// Writing clear text for field description
IF (nMemoryBank = 0) THEN
	aMemoryBank[0].sName := ' Address of last accessible memory location (read only)';
	aMemoryBank[1].sName := ' Reserved-not implemented ';
	aMemoryBank[2].sName := ' Number of last accessible memory bank (read only)';
	aMemoryBank[3].sName := ' GTIN byte 0 (MSB) (read only)';
	aMemoryBank[4].sName := ' GTIN byte 1 (read only)';
	aMemoryBank[5].sName := ' GTIN byte 2 (read only)';
	aMemoryBank[6].sName := ' GTIN byte 3 (read only)';
	aMemoryBank[7].sName := ' GTIN byte 4 (read only)';
	aMemoryBank[8].sName := ' GTIN byte 5 (LSB) (read only)';
	aMemoryBank[9].sName := ' Firmware Version (major) (read only)';
	aMemoryBank[10].sName := ' Firmware Version (m)(read only)';
	aMemoryBank[11].sName := ' Identification number byte 0 (MSB) (read only)';
	aMemoryBank[12].sName := ' Identification number byte 1 (read only)';
	aMemoryBank[13].sName := ' Identification number byte 2 (read only)';
	aMemoryBank[14].sName := ' Identification number byte 3 (read only)';
	aMemoryBank[15].sName := ' Identification number byte 4 (read only)';
	aMemoryBank[16].sName := ' Identification number byte 5 (read only)';
	aMemoryBank[17].sName := ' Identification number byte 6 (read only)';
	aMemoryBank[18].sName := ' Identification number byte 7 (LSB) (read only)';
	aMemoryBank[19].sName := ' Hardware version (major)(read only)'; 
	aMemoryBank[20].sName := ' Hardware version (minor)(read only)'; 
	aMemoryBank[21].sName := ' 101 version number (read only)';
	aMemoryBank[22].sName := ' 102 version number of all integrated control gear (read only)';
	aMemoryBank[23].sName := ' 103 version number of all integrates control devices (read only)';
	aMemoryBank[24].sName := ' Number of logical control device units in the bus unit (read only)';
	aMemoryBank[25].sName := ' Number of logical control gear units in the bus unit(read only)';
	aMemoryBank[26].sName := ' Index number of this logical control gear unit (read only)';
END_IF
IF (nMemoryBank = 1) THEN
	aMemoryBank[0].sName := ' Address of last accessible memory location (read only)';
	aMemoryBank[1].sName := ' Indicator byte (manufacturer defined) ';
	aMemoryBank[2].sName := ' Memory bank 1 lock byte';
	aMemoryBank[3].sName := ' OEM GTIN byte 0 (MSB) (read only)';
	aMemoryBank[4].sName := ' OEM GTIN byte 1 (read only)';
	aMemoryBank[5].sName := ' OEM GTIN byte 2 (read only)';
	aMemoryBank[6].sName := ' OEM GTIN byte 3 (read only)';
	aMemoryBank[7].sName := ' OEM GTIN byte 4 (read only)';
	aMemoryBank[8].sName := ' OEM GTIN byte 5 (LSB) (read only)';
	aMemoryBank[9].sName := ' OEM identification number byte 0 (MSB)';
	aMemoryBank[10].sName := ' OEM identification number byte 1';
	aMemoryBank[11].sName := ' OEM identification number byte 2';
	aMemoryBank[12].sName := ' OEM identification number byte 3';
	aMemoryBank[13].sName := ' OEM identification number byte 4';
	aMemoryBank[14].sName := ' OEM identification number byte 5';
	aMemoryBank[15].sName := ' OEM identification number byte 6';
	aMemoryBank[16].sName := ' OEM identification number byte 7 (LSB)';
END_IF
IF (nMemoryBank >= 1) THEN
	aMemoryBank[17].sName := ' Additional control gear information (lockable)';
	aMemoryBank[18].sName := ' Additional control gear information (lockable)';
	aMemoryBank[19].sName := ' Additional control gear information (lockable)';
	aMemoryBank[20].sName := ' Additional control gear information (lockable)';
	aMemoryBank[21].sName := ' Additional control gear information (lockable)';
	aMemoryBank[22].sName := ' Additional control gear information (lockable)';
	aMemoryBank[23].sName := ' Additional control gear information (lockable)';
	aMemoryBank[24].sName := ' Additional control gear information (lockable)';
	aMemoryBank[25].sName := ' Additional control gear information (lockable)';
	aMemoryBank[26].sName := ' Additional control gear information (lockable)';
	aMemoryBank[27].sName := ' Additional control gear information (lockable)';
	aMemoryBank[28].sName := ' Additional control gear information (lockable)';
	aMemoryBank[29].sName := ' Additional control gear information (lockable)';
	aMemoryBank[30].sName := ' Additional control gear information (lockable)';
	aMemoryBank[31].sName := ' Additional control gear information (lockable)';
	aMemoryBank[32].sName := ' Additional control gear information (lockable)';
	aMemoryBank[33].sName := ' Additional control gear information (lockable)';
	aMemoryBank[34].sName := ' Additional control gear information (lockable)';
	aMemoryBank[35].sName := ' Additional control gear information (lockable)';
	aMemoryBank[36].sName := ' Additional control gear information (lockable)';
	aMemoryBank[37].sName := ' Additional control gear information (lockable)';
	aMemoryBank[38].sName := ' Additional control gear information (lockable)';
	aMemoryBank[39].sName := ' Additional control gear information (lockable)';
	aMemoryBank[40].sName := ' Additional control gear information (lockable)';
	aMemoryBank[41].sName := ' Additional control gear information (lockable)';
	aMemoryBank[42].sName := ' Additional control gear information (lockable)';
	aMemoryBank[42].sName := ' Additional control gear information (lockable)';
	aMemoryBank[44].sName := ' Additional control gear information (lockable)';
	aMemoryBank[45].sName := ' Additional control gear information (lockable)';
	aMemoryBank[46].sName := ' Additional control gear information (lockable)';
	aMemoryBank[47].sName := ' Additional control gear information (lockable)';
	aMemoryBank[48].sName := ' Additional control gear information (lockable)';
	aMemoryBank[49].sName := ' Additional control gear information (lockable)';
	aMemoryBank[50].sName := ' Additional control gear information (lockable)';
	aMemoryBank[51].sName := ' Additional control gear information (lockable)';
	aMemoryBank[52].sName := ' Additional control gear information (lockable)';
	aMemoryBank[53].sName := ' Additional control gear information (lockable)';
	aMemoryBank[54].sName := ' Additional control gear information (lockable)';
	aMemoryBank[55].sName := ' Additional control gear information (lockable)';
	aMemoryBank[56].sName := ' Additional control gear information (lockable)';
	aMemoryBank[57].sName := ' Additional control gear information (lockable)';
	aMemoryBank[58].sName := ' Additional control gear information (lockable)';
	aMemoryBank[59].sName := ' Additional control gear information (lockable)';
	aMemoryBank[60].sName := ' Additional control gear information (lockable)';
	aMemoryBank[61].sName := ' Additional control gear information (lockable)';
	aMemoryBank[62].sName := ' Additional control gear information (lockable)';
	aMemoryBank[63].sName := ' Additional control gear information (lockable)';
	aMemoryBank[64].sName := ' Additional control gear information (lockable)';
	aMemoryBank[65].sName := ' Additional control gear information (lockable)';
	aMemoryBank[66].sName := ' Additional control gear information (lockable)';
	aMemoryBank[67].sName := ' Additional control gear information (lockable)';
	aMemoryBank[68].sName := ' Additional control gear information (lockable)';
	aMemoryBank[69].sName := ' Additional control gear information (lockable)';
	aMemoryBank[70].sName := ' Additional control gear information (lockable)';
	aMemoryBank[71].sName := ' Additional control gear information (lockable)';
	aMemoryBank[72].sName := ' Additional control gear information (lockable)';
	aMemoryBank[73].sName := ' Additional control gear information (lockable)';
	aMemoryBank[74].sName := ' Additional control gear information (lockable)';
	aMemoryBank[75].sName := ' Additional control gear information (lockable)';
	aMemoryBank[76].sName := ' Additional control gear information (lockable)';
	aMemoryBank[77].sName := ' Additional control gear information (lockable)';
	aMemoryBank[78].sName := ' Additional control gear information (lockable)';
	aMemoryBank[79].sName := ' Additional control gear information (lockable)';
	aMemoryBank[80].sName := ' Additional control gear information (lockable)';
	aMemoryBank[81].sName := ' Additional control gear information (lockable)';
	aMemoryBank[82].sName := ' Additional control gear information (lockable)';
	aMemoryBank[83].sName := ' Additional control gear information (lockable)';
	aMemoryBank[84].sName := ' Additional control gear information (lockable)';
	aMemoryBank[85].sName := ' Additional control gear information (lockable)';
	aMemoryBank[86].sName := ' Additional control gear information (lockable)';
	aMemoryBank[87].sName := ' Additional control gear information (lockable)';
	aMemoryBank[88].sName := ' Additional control gear information (lockable)';
	aMemoryBank[89].sName := ' Additional control gear information (lockable)';
	aMemoryBank[90].sName := ' Additional control gear information (lockable)';
	aMemoryBank[91].sName := ' Additional control gear information (lockable)';
	aMemoryBank[92].sName := ' Additional control gear information (lockable)';
	aMemoryBank[93].sName := ' Additional control gear information (lockable)';
	aMemoryBank[94].sName := ' Additional control gear information (lockable)';
	aMemoryBank[95].sName := ' Additional control gear information (lockable)';
	aMemoryBank[96].sName := ' Additional control gear information (lockable)';
	aMemoryBank[97].sName := ' Additional control gear information (lockable)';
	aMemoryBank[98].sName := ' Additional control gear information (lockable)';
	aMemoryBank[99].sName := ' Additional control gear information (lockable)';
	aMemoryBank[100].sName := ' Additional control gear information (lockable)';
	aMemoryBank[101].sName := ' Additional control gear information (lockable)';
	aMemoryBank[102].sName := ' Additional control gear information (lockable)';
	aMemoryBank[103].sName := ' Additional control gear information (lockable)';
	aMemoryBank[104].sName := ' Additional control gear information (lockable)';
	aMemoryBank[105].sName := ' Additional control gear information (lockable)';
	aMemoryBank[106].sName := ' Additional control gear information (lockable)';
	aMemoryBank[107].sName := ' Additional control gear information (lockable)';
	aMemoryBank[108].sName := ' Additional control gear information (lockable)';
	aMemoryBank[109].sName := ' Additional control gear information (lockable)';
	aMemoryBank[110].sName := ' Additional control gear information (lockable)';
	aMemoryBank[111].sName := ' Additional control gear information (lockable)';
	aMemoryBank[112].sName := ' Additional control gear information (lockable)';
	aMemoryBank[113].sName := ' Additional control gear information (lockable)';
	aMemoryBank[114].sName := ' Additional control gear information (lockable)';
	aMemoryBank[115].sName := ' Additional control gear information (lockable)';
	aMemoryBank[116].sName := ' Additional control gear information (lockable)';
	aMemoryBank[117].sName := ' Additional control gear information (lockable)';
	aMemoryBank[118].sName := ' Additional control gear information (lockable)';
	aMemoryBank[119].sName := ' Additional control gear information (lockable)';
	aMemoryBank[120].sName := ' Additional control gear information (lockable)';
	aMemoryBank[121].sName := ' Additional control gear information (lockable)';
	aMemoryBank[122].sName := ' Additional control gear information (lockable)';
	aMemoryBank[123].sName := ' Additional control gear information (lockable)';
	aMemoryBank[124].sName := ' Additional control gear information (lockable)';
	aMemoryBank[125].sName := ' Additional control gear information (lockable)';
	aMemoryBank[126].sName := ' Additional control gear information (lockable)';
	aMemoryBank[127].sName := ' Additional control gear information (lockable)';
	aMemoryBank[128].sName := ' Additional control gear information (lockable)';
	aMemoryBank[129].sName := ' Additional control gear information (lockable)';
	aMemoryBank[130].sName := ' Additional control gear information (lockable)';
	aMemoryBank[131].sName := ' Additional control gear information (lockable)';
	aMemoryBank[132].sName := ' Additional control gear information (lockable)';
	aMemoryBank[133].sName := ' Additional control gear information (lockable)';
	aMemoryBank[134].sName := ' Additional control gear information (lockable)';
	aMemoryBank[135].sName := ' Additional control gear information (lockable)';
	aMemoryBank[136].sName := ' Additional control gear information (lockable)';
	aMemoryBank[137].sName := ' Additional control gear information (lockable)';
	aMemoryBank[138].sName := ' Additional control gear information (lockable)';
	aMemoryBank[139].sName := ' Additional control gear information (lockable)';
	aMemoryBank[140].sName := ' Additional control gear information (lockable)';
	aMemoryBank[141].sName := ' Additional control gear information (lockable)';
	aMemoryBank[142].sName := ' Additional control gear information (lockable)';
	aMemoryBank[143].sName := ' Additional control gear information (lockable)';
	aMemoryBank[144].sName := ' Additional control gear information (lockable)';
	aMemoryBank[145].sName := ' Additional control gear information (lockable)';
	aMemoryBank[146].sName := ' Additional control gear information (lockable)';
	aMemoryBank[147].sName := ' Additional control gear information (lockable)';
	aMemoryBank[148].sName := ' Additional control gear information (lockable)';
	aMemoryBank[149].sName := ' Additional control gear information (lockable)';
	aMemoryBank[150].sName := ' Additional control gear information (lockable)';
	aMemoryBank[151].sName := ' Additional control gear information (lockable)';
	aMemoryBank[152].sName := ' Additional control gear information (lockable)';
	aMemoryBank[153].sName := ' Additional control gear information (lockable)';
	aMemoryBank[154].sName := ' Additional control gear information (lockable)';
	aMemoryBank[155].sName := ' Additional control gear information (lockable)';
	aMemoryBank[156].sName := ' Additional control gear information (lockable)';
	aMemoryBank[157].sName := ' Additional control gear information (lockable)';
	aMemoryBank[158].sName := ' Additional control gear information (lockable)';
	aMemoryBank[159].sName := ' Additional control gear information (lockable)';
	aMemoryBank[160].sName := ' Additional control gear information (lockable)';
	aMemoryBank[161].sName := ' Additional control gear information (lockable)';
	aMemoryBank[162].sName := ' Additional control gear information (lockable)';
	aMemoryBank[163].sName := ' Additional control gear information (lockable)';
	aMemoryBank[164].sName := ' Additional control gear information (lockable)';
	aMemoryBank[165].sName := ' Additional control gear information (lockable)';
	aMemoryBank[166].sName := ' Additional control gear information (lockable)';
	aMemoryBank[167].sName := ' Additional control gear information (lockable)';
	aMemoryBank[168].sName := ' Additional control gear information (lockable)';
	aMemoryBank[169].sName := ' Additional control gear information (lockable)';
	aMemoryBank[170].sName := ' Additional control gear information (lockable)';
	aMemoryBank[171].sName := ' Additional control gear information (lockable)';
	aMemoryBank[172].sName := ' Additional control gear information (lockable)';
	aMemoryBank[173].sName := ' Additional control gear information (lockable)';
	aMemoryBank[174].sName := ' Additional control gear information (lockable)';
	aMemoryBank[175].sName := ' Additional control gear information (lockable)';
	aMemoryBank[176].sName := ' Additional control gear information (lockable)';
	aMemoryBank[177].sName := ' Additional control gear information (lockable)';
	aMemoryBank[178].sName := ' Additional control gear information (lockable)';
	aMemoryBank[179].sName := ' Additional control gear information (lockable)';
	aMemoryBank[180].sName := ' Additional control gear information (lockable)';
	aMemoryBank[181].sName := ' Additional control gear information (lockable)';
	aMemoryBank[182].sName := ' Additional control gear information (lockable)';
	aMemoryBank[183].sName := ' Additional control gear information (lockable)';
	aMemoryBank[184].sName := ' Additional control gear information (lockable)';
	aMemoryBank[185].sName := ' Additional control gear information (lockable)';
	aMemoryBank[186].sName := ' Additional control gear information (lockable)';
	aMemoryBank[187].sName := ' Additional control gear information (lockable)';
	aMemoryBank[188].sName := ' Additional control gear information (lockable)';
	aMemoryBank[189].sName := ' Additional control gear information (lockable)';
	aMemoryBank[190].sName := ' Additional control gear information (lockable)';
	aMemoryBank[191].sName := ' Additional control gear information (lockable)';
	aMemoryBank[192].sName := ' Additional control gear information (lockable)';
	aMemoryBank[193].sName := ' Additional control gear information (lockable)';
	aMemoryBank[194].sName := ' Additional control gear information (lockable)';
	aMemoryBank[195].sName := ' Additional control gear information (lockable)';
	aMemoryBank[196].sName := ' Additional control gear information (lockable)';
	aMemoryBank[197].sName := ' Additional control gear information (lockable)';
	aMemoryBank[198].sName := ' Additional control gear information (lockable)';
	aMemoryBank[199].sName := ' Additional control gear information (lockable)';
	aMemoryBank[200].sName := ' Additional control gear information (lockable)';
	aMemoryBank[201].sName := ' Additional control gear information (lockable)';
	aMemoryBank[202].sName := ' Additional control gear information (lockable)';
	aMemoryBank[203].sName := ' Additional control gear information (lockable)';
	aMemoryBank[204].sName := ' Additional control gear information (lockable)';
	aMemoryBank[205].sName := ' Additional control gear information (lockable)';
	aMemoryBank[206].sName := ' Additional control gear information (lockable)';
	aMemoryBank[207].sName := ' Additional control gear information (lockable)';
	aMemoryBank[208].sName := ' Additional control gear information (lockable)';
	aMemoryBank[209].sName := ' Additional control gear information (lockable)';
	aMemoryBank[210].sName := ' Additional control gear information (lockable)';
	aMemoryBank[211].sName := ' Additional control gear information (lockable)';
	aMemoryBank[212].sName := ' Additional control gear information (lockable)';
	aMemoryBank[213].sName := ' Additional control gear information (lockable)';
	aMemoryBank[214].sName := ' Additional control gear information (lockable)';
	aMemoryBank[215].sName := ' Additional control gear information (lockable)';
	aMemoryBank[216].sName := ' Additional control gear information (lockable)';
	aMemoryBank[217].sName := ' Additional control gear information (lockable)';
	aMemoryBank[218].sName := ' Additional control gear information (lockable)';
	aMemoryBank[219].sName := ' Additional control gear information (lockable)';
	aMemoryBank[220].sName := ' Additional control gear information (lockable)';
	aMemoryBank[221].sName := ' Additional control gear information (lockable)';
	aMemoryBank[222].sName := ' Additional control gear information (lockable)';
	aMemoryBank[223].sName := ' Additional control gear information (lockable)';
	aMemoryBank[224].sName := ' Additional control gear information (lockable)';
	aMemoryBank[225].sName := ' Additional control gear information (lockable)';
	aMemoryBank[226].sName := ' Additional control gear information (lockable)';
	aMemoryBank[227].sName := ' Additional control gear information (lockable)';
	aMemoryBank[228].sName := ' Additional control gear information (lockable)';
	aMemoryBank[229].sName := ' Additional control gear information (lockable)';
	aMemoryBank[230].sName := ' Additional control gear information (lockable)';
	aMemoryBank[231].sName := ' Additional control gear information (lockable)';
	aMemoryBank[232].sName := ' Additional control gear information (lockable)';
	aMemoryBank[233].sName := ' Additional control gear information (lockable)';
	aMemoryBank[234].sName := ' Additional control gear information (lockable)';
	aMemoryBank[235].sName := ' Additional control gear information (lockable)';
	aMemoryBank[236].sName := ' Additional control gear information (lockable)';
	aMemoryBank[237].sName := ' Additional control gear information (lockable)';
	aMemoryBank[238].sName := ' Additional control gear information (lockable)';
	aMemoryBank[239].sName := ' Additional control gear information (lockable)';
	aMemoryBank[240].sName := ' Additional control gear information (lockable)';
	aMemoryBank[241].sName := ' Additional control gear information (lockable)';
	aMemoryBank[242].sName := ' Additional control gear information (lockable)';
	aMemoryBank[243].sName := ' Additional control gear information (lockable)';
	aMemoryBank[244].sName := ' Additional control gear information (lockable)';
	aMemoryBank[245].sName := ' Additional control gear information (lockable)';
	aMemoryBank[246].sName := ' Additional control gear information (lockable)';
	aMemoryBank[247].sName := ' Additional control gear information (lockable)';
	aMemoryBank[248].sName := ' Additional control gear information (lockable)';
	aMemoryBank[249].sName := ' Additional control gear information (lockable)';
	aMemoryBank[250].sName := ' Additional control gear information (lockable)';
	aMemoryBank[251].sName := ' Additional control gear information (lockable)';
	aMemoryBank[252].sName := ' Additional control gear information (lockable)';
	aMemoryBank[253].sName := ' Additional control gear information (lockable)';
	aMemoryBank[254].sName := ' Additional control gear information (lockable)';
END_IF
IF (nMemoryBank >= 2) THEN
	aMemoryBank[0].sName := ' Address of last accessible memory location (read only)';
	aMemoryBank[1].sName := ' Indicator byte (manufacturer defined) ';
	aMemoryBank[2].sName := ' Memory bank lock byte';
	aMemoryBank[3].sName := ' Additional control gear information (lockable)';
	aMemoryBank[4].sName := ' Additional control gear information (lockable)';
	aMemoryBank[5].sName := ' Additional control gear information (lockable)';
	aMemoryBank[6].sName := ' Additional control gear information (lockable)';
	aMemoryBank[7].sName := ' Additional control gear information (lockable)';
	aMemoryBank[8].sName := ' Additional control gear information (lockable)';
	aMemoryBank[9].sName := ' Additional control gear information (lockable)';
	aMemoryBank[10].sName := ' Additional control gear information (lockable)';
	aMemoryBank[11].sName := ' Additional control gear information (lockable)';
	aMemoryBank[12].sName := ' Additional control gear information (lockable)';
	aMemoryBank[13].sName := ' Additional control gear information (lockable)';
	aMemoryBank[14].sName := ' Additional control gear information (lockable)';
	aMemoryBank[15].sName := ' Additional control gear information (lockable)';
	aMemoryBank[16].sName := ' Additional control gear information (lockable)'; 
END_IF

END_FUNCTION_BLOCK

// ---- Tc3_DALI_PLC_Commissioning_Tool/POUs/DALI_PLC_Commissioning/FB_Part103MemoryPages.TcPOU
FUNCTION_BLOCK FB_Part103MemoryPages
VAR_INPUT
	ipDALICommunication				:	I_DALICommunication;
END_VAR
VAR_OUTPUT
	bBusy							:	BOOL;
END_VAR
VAR
	{region "Visu"}
	bRead							:	BOOL;
	bWrite							:	BOOL;
	bHideWaitSymbol					:	BOOL := TRUE;
	aMemoryBank						:	ARRAY [0..254] OF ST_DALIMemoryBank;
	{endregion}
	aValues							:	ARRAY [0..254] OF BYTE;
	nStep							:	INT;
	nAddress						:	BYTE;
	nMemoryBank						:	BYTE;
	nOffset							:	INT := 0;
	aNoValue						:	ARRAY [0..254] OF BOOL;
	nNoValue						:	BYTE;

	fb103StartQuiescentMode			:	FB_DALI103StartQuiescentMode(0);
	fb103StopQuiescentMode			:	FB_DALI103StopQuiescentMode(0);
	fb103ReadMemoryLocation			:	FB_DALI103ReadMemoryLocation(0);
	fb103WriteMemoryLocationNoReply	:	FB_DALI103WriteMemoryLocationNoReply(0);
END_VAR

IF (bRead AND (nStep = 0)) THEN
	nStep := 5;
	bRead := FALSE;
	bHideWaitSymbol := FALSE;
END_IF

IF (bWrite AND (nStep = 0)) THEN
	nStep := 1000;
	bWrite := FALSE;
	bHideWaitSymbol := FALSE;
END_IF

{region "Manage Dialog Selection}
IF (nStep = 0) THEN
	bBusy := FALSE;
ELSE
	bBusy := TRUE;
END_IF
{endregion}

{region "Execute Commands"}
CASE nStep OF
0:
{region "Init"}
	bRead := FALSE;
	bWrite := FALSE;
	bHideWaitSymbol := TRUE;

	fb103StartQuiescentMode.ipDALICommunication := ipDALICommunication;
	fb103StopQuiescentMode.ipDALICommunication := ipDALICommunication;
	fb103ReadMemoryLocation.ipDALICommunication := ipDALICommunication;
	fb103WriteMemoryLocationNoReply.ipDALICommunication := ipDALICommunication;
{endregion}
{region "Read"}
5:
{region "Start Qiescent Mode"}
	fb103StartQuiescentMode(bStart := TRUE,
							nAddress := nAddress,
							eAddressType := Tc3_DALI.E_DALIAddressType.Short,
							eCommandPriority := Tc3_DALI.E_DALICommandPriority.Middle);
	IF (NOT fb103StartQuiescentMode.bBusy) THEN
		fb103StartQuiescentMode(bStart:= FALSE);
		nStep := 10;
	END_IF
{endregion}
10:
{region "Read values from selected memory bank"}
	fb103ReadMemoryLocation(bStart := TRUE,
							nAddress := nAddress,
							eAddressType := Tc3_DALI.E_DALIAddressType.Short,
							eCommandPriority := Tc3_DALI.E_DALICommandPriority.Middle,
							nMemoryBank := nMemoryBank,
							nOffset := INT_TO_BYTE(nOffset),
							nValue=> aValues[nOffset]);
	IF (NOT fb103ReadMemoryLocation.bBusy) THEN
		aMemoryBank[nOffset].nValueDec := aValues[nOffset];
		aMemoryBank[nOffset].nValueHex := CONCAT ('0x', BYTE_TO_HEXSTR(aValues[nOffset], 2, FALSE));
		nOffset	:= nOffset+1;
		IF (nOffset > aValues[0]) THEN
			nOffset := 0;
			nStep := 20;
		END_IF
		fb103ReadMemoryLocation(bStart := FALSE);
	END_IF
{endregion}
20:
{region "Hide unused rows in table"}
	FOR nNoValue := (aValues[0] + 1) TO 254 DO
		aNoValue[nNoValue] := TRUE;
	END_FOR
	FOR nNoValue := 0 TO (aValues[0]) DO
		aNoValue[nNoValue] := FALSE;
	END_FOR
nStep := 30;
{endregion}
30:
{region "Stop Qiescent Mode"}
	fb103StopQuiescentMode(bStart:= TRUE,
						   nAddress:= nAddress,
						   eAddressType:= Tc3_DALI.E_DALIAddressType.Short,
						   eCommandPriority:= Tc3_DALI.E_DALICommandPriority.Middle);
	IF (NOT fb103StopQuiescentMode.bBusy) THEN
		fb103StopQuiescentMode(bStart := FALSE);
		nStep := 0;
	END_IF
{endregion}

1000:
{region "Change Value"}
	IF (nMemoryBank >= 1) THEN
	aValues[nOffset] := aMemoryBank[nOffset].nValueDec;
	fb103WriteMemoryLocationNoReply(bStart := TRUE,
									nAddress := nAddress,
									eAddressType := Tc3_DALI.E_DALIAddressType.Short,
									eCommandPriority := Tc3_DALI.E_DALICommandPriority.Middle,
									nMemoryBank := nMemoryBank,
									nOffset := INT_TO_BYTE(nOffset),
									nValue := aValues[nOffset]);
	IF (NOT fb103WriteMemoryLocationNoReply.bBusy) THEN
		nStep := 1010;
		fb103WriteMemoryLocationNoReply(bStart := FALSE);
	END_IF
ELSE 
	 nStep := 0;
END_IF
{endregion}
1010:
{region "read changed value"}
	 fb103ReadMemoryLocation(bStart := TRUE,
							 nAddress := nAddress,
							 eAddressType := Tc3_DALI.E_DALIAddressType.Short,
							 eCommandPriority := Tc3_DALI.E_DALICommandPriority.Middle,
							 nMemoryBank := nMemoryBank,
							 nOffset := INT_TO_BYTE(nOffset),
							 nValue=> aValues[nOffset]);
	IF (NOT fb103ReadMemoryLocation.bBusy) THEN
		aMemoryBank[nOffset].nValueDec := aValues[nOffset];
		aMemoryBank[nOffset].nValueHex := CONCAT ('0x', BYTE_TO_HEXSTR(aValues[nOffset], 2, FALSE));
		nStep := 0;
		fb103ReadMemoryLocation(bStart := FALSE);
	END_IF
{endregion}
END_CASE

// Filling the according fields of the Array Memory Bank for the HMI display
// Writing clear text for offset description
aMemoryBank[0].sOffset := '0 (0x00)';
aMemoryBank[1].sOffset := '1 (0x01)';
aMemoryBank[2].sOffset := '2 (0x02)';
aMemoryBank[3].sOffset := '3 (0x03)';
aMemoryBank[4].sOffset := '4 (0x04)';
aMemoryBank[5].sOffset := '5 (0x05)';
aMemoryBank[6].sOffset := '6 (0x06)';
aMemoryBank[7].sOffset := '7 (0x07)';
aMemoryBank[8].sOffset := '8 (0x08)';
aMemoryBank[9].sOffset := '9 (0x09)';
aMemoryBank[10].sOffset := '10 (0x0A)';
aMemoryBank[11].sOffset := '11 (0x0B)';
aMemoryBank[12].sOffset := '12 (0x0C)';
aMemoryBank[13].sOffset := '13 (0x0D)';
aMemoryBank[14].sOffset := '14 (0x0E)';
aMemoryBank[15].sOffset := '15 (0x0F)';
aMemoryBank[16].sOffset := '16 (0x10)';
aMemoryBank[17].sOffset := '17 (0x11)';
aMemoryBank[18].sOffset := '18 (0x12)';
aMemoryBank[19].sOffset := '19 (0x13)';
aMemoryBank[20].sOffset := '20 (0x14)';
aMemoryBank[21].sOffset := '21 (0x15)';
aMemoryBank[22].sOffset := '22 (0x16)';
aMemoryBank[23].sOffset := '23 (0x17)';
aMemoryBank[24].sOffset := '24 (0x18)';
aMemoryBank[25].sOffset := '25 (0x19)';
aMemoryBank[26].sOffset := '26 (0x1A)';
aMemoryBank[27].sOffset := '27 (0x1B)';
aMemoryBank[28].sOffset := '28 (0x1C)';
aMemoryBank[29].sOffset := '29 (0x1D)';
aMemoryBank[30].sOffset := '30 (0x1E)';
aMemoryBank[31].sOffset := '31 (0x1F)';
aMemoryBank[32].sOffset := '32 (0x20)';
aMemoryBank[33].sOffset := '33 (0x21)';
aMemoryBank[34].sOffset := '34 (0x22)';
aMemoryBank[35].sOffset := '35 (0x23)';
aMemoryBank[36].sOffset := '36 (0x24)';
aMemoryBank[37].sOffset := '37 (0x25)';
aMemoryBank[38].sOffset := '38 (0x26)';
aMemoryBank[39].sOffset := '39 (0x27)';
aMemoryBank[40].sOffset := '40 (0x28)';
aMemoryBank[41].sOffset := '41 (0x29)';
aMemoryBank[42].sOffset := '42 (0x2A)';
aMemoryBank[42].sOffset := '43 (0x2B)';
aMemoryBank[44].sOffset := '44 (0x2C)';
aMemoryBank[45].sOffset := '45 (0x2D)';
aMemoryBank[46].sOffset := '46 (0x2E)';
aMemoryBank[47].sOffset := '47 (0x2F)';
aMemoryBank[48].sOffset := '48 (0x30)';
aMemoryBank[49].sOffset := '49 (0x31)';
aMemoryBank[50].sOffset := '50 (0x32)';
aMemoryBank[51].sOffset := '51 (0x33)';
aMemoryBank[52].sOffset := '52 (0x34)';
aMemoryBank[53].sOffset := '53 (0x35)';
aMemoryBank[54].sOffset := '54 (0x36)';
aMemoryBank[55].sOffset := '55 (0x37)';
aMemoryBank[56].sOffset := '56 (0x38)';
aMemoryBank[57].sOffset := '57 (0x39)';
aMemoryBank[58].sOffset := '58 (0x3A)';
aMemoryBank[59].sOffset := '59 (0x3B)';
aMemoryBank[60].sOffset := '60 (0x3C)';
aMemoryBank[61].sOffset := '61 (0x3D)';
aMemoryBank[62].sOffset := '62 (0x3F)';
aMemoryBank[63].sOffset := '63 (0x3D)';
aMemoryBank[64].sOffset := '64 (0x40)';
aMemoryBank[65].sOffset := '65 (0x41)';
aMemoryBank[66].sOffset := '66 (0x42)';
aMemoryBank[67].sOffset := '67 (0x43)';
aMemoryBank[68].sOffset := '68 (0x44)';
aMemoryBank[69].sOffset := '69 (0x45)';
aMemoryBank[70].sOffset := '70 (0x46)';
aMemoryBank[71].sOffset := '71 (0x47)';
aMemoryBank[72].sOffset := '72 (0x48)';
aMemoryBank[73].sOffset := '73 (0x49)';
aMemoryBank[74].sOffset := '74 (0x4A)';
aMemoryBank[75].sOffset := '75 (0x4B)';
aMemoryBank[76].sOffset := '76 (0x4C)';
aMemoryBank[77].sOffset := '77 (0x4D)';
aMemoryBank[78].sOffset := '78 (0x4E)';
aMemoryBank[79].sOffset := '79 (0x4F)';
aMemoryBank[80].sOffset := '80 (0x50)';
aMemoryBank[81].sOffset := '81 (0x51)';
aMemoryBank[82].sOffset := '82 (0x52)';
aMemoryBank[83].sOffset := '83 (0x53)';
aMemoryBank[84].sOffset := '84 (0x54)';
aMemoryBank[85].sOffset := '85 (0x55)';
aMemoryBank[86].sOffset := '86 (0x56)';
aMemoryBank[87].sOffset := '87 (0x57)';
aMemoryBank[88].sOffset := '88 (0x58)';
aMemoryBank[89].sOffset := '89 (0x59)';
aMemoryBank[90].sOffset := '90 (0x5A)';
aMemoryBank[91].sOffset := '91 (0x5B)';
aMemoryBank[92].sOffset := '92 (0x5C)';
aMemoryBank[93].sOffset := '93 (0x5D)';
aMemoryBank[94].sOffset := '94 (0x5E)';
aMemoryBank[95].sOffset := '95 (0x5F)';
aMemoryBank[96].sOffset := '96 (0x60)';
aMemoryBank[97].sOffset := '97 (0x61)';
aMemoryBank[98].sOffset := '98 (0x62)';
aMemoryBank[99].sOffset := '99 (0x63)';
aMemoryBank[100].sOffset := '100 (0x64)';
aMemoryBank[101].sOffset := '101 (0x65)';
aMemoryBank[102].sOffset := '102 (0x66)';
aMemoryBank[103].sOffset := '103 (0x67)';
aMemoryBank[104].sOffset := '104 (0x68)';
aMemoryBank[105].sOffset := '105 (0x69)';
aMemoryBank[106].sOffset := '106 (0x6A)';
aMemoryBank[107].sOffset := '107 (0x6B)';
aMemoryBank[108].sOffset := '108 (0x6C)';
aMemoryBank[109].sOffset := '109 (0x6D)';
aMemoryBank[110].sOffset := '110 (0x6E)';
aMemoryBank[111].sOffset := '111 (0x6F)';
aMemoryBank[112].sOffset := '112 (0x70)';
aMemoryBank[113].sOffset := '113 (0x71)';
aMemoryBank[114].sOffset := '114 (0x72)';
aMemoryBank[115].sOffset := '115 (0x73)';
aMemoryBank[116].sOffset := '116 (0x74)';
aMemoryBank[117].sOffset := '117 (0x75)';
aMemoryBank[118].sOffset := '118 (0x76)';
aMemoryBank[119].sOffset := '119 (0x77)';
aMemoryBank[120].sOffset := '120 (0x78)';
aMemoryBank[121].sOffset := '121 (0x79)';
aMemoryBank[122].sOffset := '122 (0x7A)';
aMemoryBank[123].sOffset := '123 (0x7B)';
aMemoryBank[124].sOffset := '124 (0x7C)';
aMemoryBank[125].sOffset := '125 (0x7D)';
aMemoryBank[126].sOffset := '126 (0x7E)';
aMemoryBank[127].sOffset := '127 (0x7F)';
aMemoryBank[128].sOffset := '128 (0x80)';
aMemoryBank[129].sOffset := '129 (0x81)';
aMemoryBank[130].sOffset := '130 (0x82)';
aMemoryBank[131].sOffset := '131 (0x83)';
aMemoryBank[132].sOffset := '132 (0x84)';
aMemoryBank[133].sOffset := '133 (0x85)';
aMemoryBank[134].sOffset := '134 (0x86)';
aMemoryBank[135].sOffset := '135 (0x87)';
aMemoryBank[136].sOffset := '136 (0x88)';
aMemoryBank[137].sOffset := '137 (0x89)';
aMemoryBank[138].sOffset := '138 (0x8A)';
aMemoryBank[139].sOffset := '139 (0x8B)';
aMemoryBank[140].sOffset := '140 (0x8C)';
aMemoryBank[141].sOffset := '141 (0x8D)';
aMemoryBank[142].sOffset := '142 (0x8E)';
aMemoryBank[143].sOffset := '143 (0x8F)';
aMemoryBank[144].sOffset := '144 (0x90)';
aMemoryBank[145].sOffset := '145 (0x91)';
aMemoryBank[146].sOffset := '146 (0x92)';
aMemoryBank[147].sOffset := '147 (0x93)';
aMemoryBank[148].sOffset := '148 (0x94)';
aMemoryBank[149].sOffset := '149 (0x95)';
aMemoryBank[150].sOffset := '150 (0x96)';
aMemoryBank[151].sOffset := '151 (0x97)';
aMemoryBank[152].sOffset := '152 (0x98)';
aMemoryBank[153].sOffset := '153 (0x99)';
aMemoryBank[154].sOffset := '154 (0x9A)';
aMemoryBank[155].sOffset := '155 (0x9B)';
aMemoryBank[156].sOffset := '156 (0x9C)';
aMemoryBank[157].sOffset := '157 (0x9D)';
aMemoryBank[158].sOffset := '158 (0x9E)';
aMemoryBank[159].sOffset := '159 (0x9F)';
aMemoryBank[160].sOffset := '160 (0xA0)';
aMemoryBank[161].sOffset := '161 (0xA1)';
aMemoryBank[162].sOffset := '162 (0xA2)';
aMemoryBank[163].sOffset := '163 (0xA3)';
aMemoryBank[164].sOffset := '164 (0xA4)';
aMemoryBank[165].sOffset := '165 (0xA5)';
aMemoryBank[166].sOffset := '166 (0xA6)';
aMemoryBank[167].sOffset := '167 (0xA7)';
aMemoryBank[168].sOffset := '168 (0xA8)';
aMemoryBank[169].sOffset := '169 (0xA9)';
aMemoryBank[170].sOffset := '170 (0xAA)';
aMemoryBank[171].sOffset := '171 (0xAB)';
aMemoryBank[172].sOffset := '172 (0xAC)';
aMemoryBank[173].sOffset := '173 (0xAD)';
aMemoryBank[174].sOffset := '174 (0xAE)';
aMemoryBank[175].sOffset := '175 (0xAF)';
aMemoryBank[176].sOffset := '176 (0xB0)';
aMemoryBank[177].sOffset := '177 (0xB1)';
aMemoryBank[178].sOffset := '178 (0xB2)';
aMemoryBank[179].sOffset := '179 (0xB3)';
aMemoryBank[180].sOffset := '180 (0xB4)';
aMemoryBank[181].sOffset := '181 (0xB5)';
aMemoryBank[182].sOffset := '182 (0xB6)';
aMemoryBank[183].sOffset := '183 (0xB7)';
aMemoryBank[184].sOffset := '184 (0xB8)';
aMemoryBank[185].sOffset := '185 (0xB9)';
aMemoryBank[186].sOffset := '186 (0xBA)';
aMemoryBank[187].sOffset := '187 (0xBB)';
aMemoryBank[188].sOffset := '188 (0xBC)';
aMemoryBank[189].sOffset := '189 (0xBD)';
aMemoryBank[190].sOffset := '190 (0xDE)';
aMemoryBank[191].sOffset := '191 (0xBF)';
aMemoryBank[192].sOffset := '192 (0xC0)';
aMemoryBank[193].sOffset := '193 (0xC1)';
aMemoryBank[194].sOffset := '194 (0xC3)';
aMemoryBank[195].sOffset := '195 (0xC4)';
aMemoryBank[196].sOffset := '196 (0xC5)';
aMemoryBank[197].sOffset := '197 (0xC6)';
aMemoryBank[198].sOffset := '198 (0xC7)';
aMemoryBank[199].sOffset := '199 (0xC8)';
aMemoryBank[200].sOffset := '200 (0xC9)';
aMemoryBank[201].sOffset := '201 (0xCA)';
aMemoryBank[202].sOffset := '202 (0xCB)';
aMemoryBank[203].sOffset := '203 (0xCC)';
aMemoryBank[204].sOffset := '204 (0xCD)';
aMemoryBank[205].sOffset := '205 (0xCE)';
aMemoryBank[206].sOffset := '206 (0xCF)';
aMemoryBank[207].sOffset := '207 (0xD0)';
aMemoryBank[208].sOffset := '208 (0xD1)';
aMemoryBank[209].sOffset := '209 (0xD2)';
aMemoryBank[210].sOffset := '210 (0xD3)';
aMemoryBank[211].sOffset := '211 (0xD4)';
aMemoryBank[212].sOffset := '212 (0xD5)';
aMemoryBank[213].sOffset := '213 (0xD6)';
aMemoryBank[214].sOffset := '214 (0xD7)';
aMemoryBank[215].sOffset := '215 (0xD8)';
aMemoryBank[216].sOffset := '216 (0xD9)';
aMemoryBank[217].sOffset := '217 (0xDA)';
aMemoryBank[218].sOffset := '218 (0xDB)';
aMemoryBank[219].sOffset := '219 (0xDC)';
aMemoryBank[220].sOffset := '220 (0xDD)';
aMemoryBank[221].sOffset := '221 (0xDE)';
aMemoryBank[222].sOffset := '222 (0xDF)';
aMemoryBank[223].sOffset := '223 (0xE0)';
aMemoryBank[224].sOffset := '224 (0xE1)';
aMemoryBank[225].sOffset := '225 (0xE2)';
aMemoryBank[226].sOffset := '226 (0xE3)';
aMemoryBank[227].sOffset := '227 (0xE4)';
aMemoryBank[228].sOffset := '228 (0xE5)';
aMemoryBank[229].sOffset := '229 (0xE6)';
aMemoryBank[230].sOffset := '230 (0xE7)';
aMemoryBank[231].sOffset := '231 (0xE8)';
aMemoryBank[232].sOffset := '232 (0xE9)';
aMemoryBank[233].sOffset := '233 (0xEA)';
aMemoryBank[234].sOffset := '234 (0xEB)';
aMemoryBank[235].sOffset := '235 (0xEC)';
aMemoryBank[236].sOffset := '236 (0xED)';
aMemoryBank[237].sOffset := '237 (0xEE)';
aMemoryBank[238].sOffset := '238 (0xEF)';
aMemoryBank[239].sOffset := '239 (0xF0)';
aMemoryBank[240].sOffset := '240 (0xF1)';
aMemoryBank[241].sOffset := '241 (0xF2)';
aMemoryBank[242].sOffset := '242 (0xF3)';
aMemoryBank[243].sOffset := '243 (0xF4)';
aMemoryBank[244].sOffset := '244 (0xF5)';
aMemoryBank[245].sOffset := '245 (0xF6)';
aMemoryBank[246].sOffset := '246 (0xF7)';
aMemoryBank[247].sOffset := '247 (0xF8)';
aMemoryBank[248].sOffset := '248 (0xF9)';
aMemoryBank[249].sOffset := '249 (0xFA)';
aMemoryBank[250].sOffset := '250 (0xFB)';
aMemoryBank[251].sOffset := '251 (0xFC)';
aMemoryBank[252].sOffset := '252 (0xFD)';
aMemoryBank[253].sOffset := '253 (0xFE)';
aMemoryBank[254].sOffset := '254 (0xFF)';

// Writing clear text for field description
IF (nMemoryBank = 0) THEN
	aMemoryBank[0].sName := ' Address of last accessible memory location (read only)';
	aMemoryBank[1].sName := ' Reserved-not implemented ';
	aMemoryBank[2].sName := ' Number of last accessible memory bank (read only)';
	aMemoryBank[3].sName := ' GTIN byte 0 (MSB) (read only)';
	aMemoryBank[4].sName := ' GTIN byte 1 (read only)';
	aMemoryBank[5].sName := ' GTIN byte 2 (read only)';
	aMemoryBank[6].sName := ' GTIN byte 3 (read only)';
	aMemoryBank[7].sName := ' GTIN byte 4 (read only)';
	aMemoryBank[8].sName := ' GTIN byte 5 (LSB) (read only)';
	aMemoryBank[9].sName := ' Firmware Version (major) (read only)';
	aMemoryBank[10].sName := ' Firmware Version (minor)(read only)';
	aMemoryBank[11].sName := ' Identification number byte 0 (MSB) (read only)';
	aMemoryBank[12].sName := ' Identification number byte 1 (read only)';
	aMemoryBank[13].sName := ' Identification number byte 2 (read only)';
	aMemoryBank[14].sName := ' Identification number byte 3 (read only)';
	aMemoryBank[15].sName := ' Identification number byte 4 (read only)';
	aMemoryBank[16].sName := ' Identification number byte 5 (read only)';
	aMemoryBank[17].sName := ' Identification number byte 6 (read only)';
	aMemoryBank[18].sName := ' Identification number byte 7 (LSB) (read only)';
	aMemoryBank[19].sName := ' Hardware version (major) (read only)';
	aMemoryBank[20].sName := ' Hardware version (minor) (read only)';
	aMemoryBank[21].sName := ' 101 version number (read only)';
	aMemoryBank[22].sName := ' 102 version number of all integrated control gear (read only)';
	aMemoryBank[23].sName := ' 103 version number of all integrates control devices (read only)';
	aMemoryBank[24].sName := ' Number of logical control device units in the bus unit (read only)';
	aMemoryBank[25].sName := ' Number of logical control gear units in the bus unit (read only)';
	aMemoryBank[26].sName := ' Index number of this logical control device unit (read only)';
END_IF
IF (nMemoryBank = 1) THEN
	aMemoryBank[0].sName := ' Address of last accessible memory location (read only)';
	aMemoryBank[1].sName := ' Indicator byte (manufacturer defined) ';
	aMemoryBank[2].sName := ' Memory bank 1 lock byte';
	aMemoryBank[3].sName := ' OEM GTIN byte 0 (MSB) (read only)';
	aMemoryBank[4].sName := ' OEM GTIN byte 1 (read only)';
	aMemoryBank[5].sName := ' OEM GTIN byte 2 (read only)';
	aMemoryBank[6].sName := ' OEM GTIN byte 3 (read only)';
	aMemoryBank[7].sName := ' OEM GTIN byte 4 (read only)';
	aMemoryBank[8].sName := ' OEM GTIN byte 5 (LSB) (read only)';
	aMemoryBank[9].sName := ' OEM identification number byte 0 (MSB)';
	aMemoryBank[10].sName := ' OEM identification number byte 1';
	aMemoryBank[11].sName := ' OEM identification number byte 2';
	aMemoryBank[12].sName := ' OEM identification number byte 3';
	aMemoryBank[13].sName := ' OEM identification number byte 4';
	aMemoryBank[14].sName := ' OEM identification number byte 5';
	aMemoryBank[15].sName := ' OEM identification number byte 6';
	aMemoryBank[16].sName := ' OEM identification number byte 7 (LSB)';
END_IF
IF (nMemoryBank >= 1) THEN
	aMemoryBank[17].sName := ' Additional control device information (lockable)';
	aMemoryBank[18].sName := ' Additional control device information (lockable)';
	aMemoryBank[19].sName := ' Additional control device information (lockable)';
	aMemoryBank[20].sName := ' Additional control device information (lockable)';
	aMemoryBank[21].sName := ' Additional control device information (lockable)';
	aMemoryBank[22].sName := ' Additional control device information (lockable)';
	aMemoryBank[23].sName := ' Additional control device information (lockable)';
	aMemoryBank[24].sName := ' Additional control device information (lockable)';
	aMemoryBank[25].sName := ' Additional control device information (lockable)';
	aMemoryBank[26].sName := ' Additional control device information (lockable)';
	aMemoryBank[27].sName := ' Additional control device information (lockable)';
	aMemoryBank[28].sName := ' Additional control device information (lockable)';
	aMemoryBank[29].sName := ' Additional control device information (lockable)';
	aMemoryBank[30].sName := ' Additional control device information (lockable)';
	aMemoryBank[31].sName := ' Additional control device information (lockable)';
	aMemoryBank[32].sName := ' Additional control device information (lockable)';
	aMemoryBank[33].sName := ' Additional control device information (lockable)';
	aMemoryBank[34].sName := ' Additional control device information (lockable)';
	aMemoryBank[35].sName := ' Additional control device information (lockable)';
	aMemoryBank[36].sName := ' Additional control device information (lockable)';
	aMemoryBank[37].sName := ' Additional control device information (lockable)';
	aMemoryBank[38].sName := ' Additional control device information (lockable)';
	aMemoryBank[39].sName := ' Additional control device information (lockable)';
	aMemoryBank[40].sName := ' Additional control device information (lockable)';
	aMemoryBank[41].sName := ' Additional control device information (lockable)';
	aMemoryBank[42].sName := ' Additional control device information (lockable)';
	aMemoryBank[42].sName := ' Additional control device information (lockable)';
	aMemoryBank[44].sName := ' Additional control device information (lockable)';
	aMemoryBank[45].sName := ' Additional control device information (lockable)';
	aMemoryBank[46].sName := ' Additional control device information (lockable)';
	aMemoryBank[47].sName := ' Additional control device information (lockable)';
	aMemoryBank[48].sName := ' Additional control device information (lockable)';
	aMemoryBank[49].sName := ' Additional control device information (lockable)';
	aMemoryBank[50].sName := ' Additional control device information (lockable)';
	aMemoryBank[51].sName := ' Additional control device information (lockable)';
	aMemoryBank[52].sName := ' Additional control device information (lockable)';
	aMemoryBank[53].sName := ' Additional control device information (lockable)';
	aMemoryBank[54].sName := ' Additional control device information (lockable)';
	aMemoryBank[55].sName := ' Additional control device information (lockable)';
	aMemoryBank[56].sName := ' Additional control device information (lockable)';
	aMemoryBank[57].sName := ' Additional control device information (lockable)';
	aMemoryBank[58].sName := ' Additional control device information (lockable)';
	aMemoryBank[59].sName := ' Additional control device information (lockable)';
	aMemoryBank[60].sName := ' Additional control device information (lockable)';
	aMemoryBank[61].sName := ' Additional control device information (lockable)';
	aMemoryBank[62].sName := ' Additional control device information (lockable)';
	aMemoryBank[63].sName := ' Additional control device information (lockable)';
	aMemoryBank[64].sName := ' Additional control device information (lockable)';
	aMemoryBank[65].sName := ' Additional control device information (lockable)';
	aMemoryBank[66].sName := ' Additional control device information (lockable)';
	aMemoryBank[67].sName := ' Additional control device information (lockable)';
	aMemoryBank[68].sName := ' Additional control device information (lockable)';
	aMemoryBank[69].sName := ' Additional control device information (lockable)';
	aMemoryBank[70].sName := ' Additional control device information (lockable)';
	aMemoryBank[71].sName := ' Additional control device information (lockable)';
	aMemoryBank[72].sName := ' Additional control device information (lockable)';
	aMemoryBank[73].sName := ' Additional control device information (lockable)';
	aMemoryBank[74].sName := ' Additional control device information (lockable)';
	aMemoryBank[75].sName := ' Additional control device information (lockable)';
	aMemoryBank[76].sName := ' Additional control device information (lockable)';
	aMemoryBank[77].sName := ' Additional control device information (lockable)';
	aMemoryBank[78].sName := ' Additional control device information (lockable)';
	aMemoryBank[79].sName := ' Additional control device information (lockable)';
	aMemoryBank[80].sName := ' Additional control device information (lockable)';
	aMemoryBank[81].sName := ' Additional control device information (lockable)';
	aMemoryBank[82].sName := ' Additional control device information (lockable)';
	aMemoryBank[83].sName := ' Additional control device information (lockable)';
	aMemoryBank[84].sName := ' Additional control device information (lockable)';
	aMemoryBank[85].sName := ' Additional control device information (lockable)';
	aMemoryBank[86].sName := ' Additional control device information (lockable)';
	aMemoryBank[87].sName := ' Additional control device information (lockable)';
	aMemoryBank[88].sName := ' Additional control device information (lockable)';
	aMemoryBank[89].sName := ' Additional control device information (lockable)';
	aMemoryBank[90].sName := ' Additional control device information (lockable)';
	aMemoryBank[91].sName := ' Additional control device information (lockable)';
	aMemoryBank[92].sName := ' Additional control device information (lockable)';
	aMemoryBank[93].sName := ' Additional control device information (lockable)';
	aMemoryBank[94].sName := ' Additional control device information (lockable)';
	aMemoryBank[95].sName := ' Additional control device information (lockable)';
	aMemoryBank[96].sName := ' Additional control device information (lockable)';
	aMemoryBank[97].sName := ' Additional control device information (lockable)';
	aMemoryBank[98].sName := ' Additional control device information (lockable)';
	aMemoryBank[99].sName := ' Additional control device information (lockable)';
	aMemoryBank[100].sName := ' Additional control device information (lockable)';
	aMemoryBank[101].sName := ' Additional control device information (lockable)';
	aMemoryBank[102].sName := ' Additional control device information (lockable)';
	aMemoryBank[103].sName := ' Additional control device information (lockable)';
	aMemoryBank[104].sName := ' Additional control device information (lockable)';
	aMemoryBank[105].sName := ' Additional control device information (lockable)';
	aMemoryBank[106].sName := ' Additional control device information (lockable)';
	aMemoryBank[107].sName := ' Additional control device information (lockable)';
	aMemoryBank[108].sName := ' Additional control device information (lockable)';
	aMemoryBank[109].sName := ' Additional control device information (lockable)';
	aMemoryBank[110].sName := ' Additional control device information (lockable)';
	aMemoryBank[111].sName := ' Additional control device information (lockable)';
	aMemoryBank[112].sName := ' Additional control device information (lockable)';
	aMemoryBank[113].sName := ' Additional control device information (lockable)';
	aMemoryBank[114].sName := ' Additional control device information (lockable)';
	aMemoryBank[115].sName := ' Additional control device information (lockable)';
	aMemoryBank[116].sName := ' Additional control device information (lockable)';
	aMemoryBank[117].sName := ' Additional control device information (lockable)';
	aMemoryBank[118].sName := ' Additional control device information (lockable)';
	aMemoryBank[119].sName := ' Additional control device information (lockable)';
	aMemoryBank[120].sName := ' Additional control device information (lockable)';
	aMemoryBank[121].sName := ' Additional control device information (lockable)';
	aMemoryBank[122].sName := ' Additional control device information (lockable)';
	aMemoryBank[123].sName := ' Additional control device information (lockable)';
	aMemoryBank[124].sName := ' Additional control device information (lockable)';
	aMemoryBank[125].sName := ' Additional control device information (lockable)';
	aMemoryBank[126].sName := ' Additional control device information (lockable)';
	aMemoryBank[127].sName := ' Additional control device information (lockable)';
	aMemoryBank[128].sName := ' Additional control device information (lockable)';
	aMemoryBank[129].sName := ' Additional control device information (lockable)';
	aMemoryBank[130].sName := ' Additional control device information (lockable)';
	aMemoryBank[131].sName := ' Additional control device information (lockable)';
	aMemoryBank[132].sName := ' Additional control device information (lockable)';
	aMemoryBank[133].sName := ' Additional control device information (lockable)';
	aMemoryBank[134].sName := ' Additional control device information (lockable)';
	aMemoryBank[135].sName := ' Additional control device information (lockable)';
	aMemoryBank[136].sName := ' Additional control device information (lockable)';
	aMemoryBank[137].sName := ' Additional control device information (lockable)';
	aMemoryBank[138].sName := ' Additional control device information (lockable)';
	aMemoryBank[139].sName := ' Additional control device information (lockable)';
	aMemoryBank[140].sName := ' Additional control device information (lockable)';
	aMemoryBank[141].sName := ' Additional control device information (lockable)';
	aMemoryBank[142].sName := ' Additional control device information (lockable)';
	aMemoryBank[143].sName := ' Additional control device information (lockable)';
	aMemoryBank[144].sName := ' Additional control device information (lockable)';
	aMemoryBank[145].sName := ' Additional control device information (lockable)';
	aMemoryBank[146].sName := ' Additional control device information (lockable)';
	aMemoryBank[147].sName := ' Additional control device information (lockable)';
	aMemoryBank[148].sName := ' Additional control device information (lockable)';
	aMemoryBank[149].sName := ' Additional control device information (lockable)';
	aMemoryBank[150].sName := ' Additional control device information (lockable)';
	aMemoryBank[151].sName := ' Additional control device information (lockable)';
	aMemoryBank[152].sName := ' Additional control device information (lockable)';
	aMemoryBank[153].sName := ' Additional control device information (lockable)';
	aMemoryBank[154].sName := ' Additional control device information (lockable)';
	aMemoryBank[155].sName := ' Additional control device information (lockable)';
	aMemoryBank[156].sName := ' Additional control device information (lockable)';
	aMemoryBank[157].sName := ' Additional control device information (lockable)';
	aMemoryBank[158].sName := ' Additional control device information (lockable)';
	aMemoryBank[159].sName := ' Additional control device information (lockable)';
	aMemoryBank[160].sName := ' Additional control device information (lockable)';
	aMemoryBank[161].sName := ' Additional control device information (lockable)';
	aMemoryBank[162].sName := ' Additional control device information (lockable)';
	aMemoryBank[163].sName := ' Additional control device information (lockable)';
	aMemoryBank[164].sName := ' Additional control device information (lockable)';
	aMemoryBank[165].sName := ' Additional control device information (lockable)';
	aMemoryBank[166].sName := ' Additional control device information (lockable)';
	aMemoryBank[167].sName := ' Additional control device information (lockable)';
	aMemoryBank[168].sName := ' Additional control device information (lockable)';
	aMemoryBank[169].sName := ' Additional control device information (lockable)';
	aMemoryBank[170].sName := ' Additional control device information (lockable)';
	aMemoryBank[171].sName := ' Additional control device information (lockable)';
	aMemoryBank[172].sName := ' Additional control device information (lockable)';
	aMemoryBank[173].sName := ' Additional control device information (lockable)';
	aMemoryBank[174].sName := ' Additional control device information (lockable)';
	aMemoryBank[175].sName := ' Additional control device information (lockable)';
	aMemoryBank[176].sName := ' Additional control device information (lockable)';
	aMemoryBank[177].sName := ' Additional control device information (lockable)';
	aMemoryBank[178].sName := ' Additional control device information (lockable)';
	aMemoryBank[179].sName := ' Additional control device information (lockable)';
	aMemoryBank[180].sName := ' Additional control device information (lockable)';
	aMemoryBank[181].sName := ' Additional control device information (lockable)';
	aMemoryBank[182].sName := ' Additional control device information (lockable)';
	aMemoryBank[183].sName := ' Additional control device information (lockable)';
	aMemoryBank[184].sName := ' Additional control device information (lockable)';
	aMemoryBank[185].sName := ' Additional control device information (lockable)';
	aMemoryBank[186].sName := ' Additional control device information (lockable)';
	aMemoryBank[187].sName := ' Additional control device information (lockable)';
	aMemoryBank[188].sName := ' Additional control device information (lockable)';
	aMemoryBank[189].sName := ' Additional control device information (lockable)';
	aMemoryBank[190].sName := ' Additional control device information (lockable)';
	aMemoryBank[191].sName := ' Additional control device information (lockable)';
	aMemoryBank[192].sName := ' Additional control device information (lockable)';
	aMemoryBank[193].sName := ' Additional control device information (lockable)';
	aMemoryBank[194].sName := ' Additional control device information (lockable)';
	aMemoryBank[195].sName := ' Additional control device information (lockable)';
	aMemoryBank[196].sName := ' Additional control device information (lockable)';
	aMemoryBank[197].sName := ' Additional control device information (lockable)';
	aMemoryBank[198].sName := ' Additional control device information (lockable)';
	aMemoryBank[199].sName := ' Additional control device information (lockable)';
	aMemoryBank[200].sName := ' Additional control device information (lockable)';
	aMemoryBank[201].sName := ' Additional control device information (lockable)';
	aMemoryBank[202].sName := ' Additional control device information (lockable)';
	aMemoryBank[203].sName := ' Additional control device information (lockable)';
	aMemoryBank[204].sName := ' Additional control device information (lockable)';
	aMemoryBank[205].sName := ' Additional control device information (lockable)';
	aMemoryBank[206].sName := ' Additional control device information (lockable)';
	aMemoryBank[207].sName := ' Additional control device information (lockable)';
	aMemoryBank[208].sName := ' Additional control device information (lockable)';
	aMemoryBank[209].sName := ' Additional control device information (lockable)';
	aMemoryBank[210].sName := ' Additional control device information (lockable)';
	aMemoryBank[211].sName := ' Additional control device information (lockable)';
	aMemoryBank[212].sName := ' Additional control device information (lockable)';
	aMemoryBank[213].sName := ' Additional control device information (lockable)';
	aMemoryBank[214].sName := ' Additional control device information (lockable)';
	aMemoryBank[215].sName := ' Additional control device information (lockable)';
	aMemoryBank[216].sName := ' Additional control device information (lockable)';
	aMemoryBank[217].sName := ' Additional control device information (lockable)';
	aMemoryBank[218].sName := ' Additional control device information (lockable)';
	aMemoryBank[219].sName := ' Additional control device information (lockable)';
	aMemoryBank[220].sName := ' Additional control device information (lockable)';
	aMemoryBank[221].sName := ' Additional control device information (lockable)';
	aMemoryBank[222].sName := ' Additional control device information (lockable)';
	aMemoryBank[223].sName := ' Additional control device information (lockable)';
	aMemoryBank[224].sName := ' Additional control device information (lockable)';
	aMemoryBank[225].sName := ' Additional control device information (lockable)';
	aMemoryBank[226].sName := ' Additional control device information (lockable)';
	aMemoryBank[227].sName := ' Additional control device information (lockable)';
	aMemoryBank[228].sName := ' Additional control device information (lockable)';
	aMemoryBank[229].sName := ' Additional control device information (lockable)';
	aMemoryBank[230].sName := ' Additional control device information (lockable)';
	aMemoryBank[231].sName := ' Additional control device information (lockable)';
	aMemoryBank[232].sName := ' Additional control device information (lockable)';
	aMemoryBank[233].sName := ' Additional control device information (lockable)';
	aMemoryBank[234].sName := ' Additional control device information (lockable)';
	aMemoryBank[235].sName := ' Additional control device information (lockable)';
	aMemoryBank[236].sName := ' Additional control device information (lockable)';
	aMemoryBank[237].sName := ' Additional control device information (lockable)';
	aMemoryBank[238].sName := ' Additional control device information (lockable)';
	aMemoryBank[239].sName := ' Additional control device information (lockable)';
	aMemoryBank[240].sName := ' Additional control device information (lockable)';
	aMemoryBank[241].sName := ' Additional control device information (lockable)';
	aMemoryBank[242].sName := ' Additional control device information (lockable)';
	aMemoryBank[243].sName := ' Additional control device information (lockable)';
	aMemoryBank[244].sName := ' Additional control device information (lockable)';
	aMemoryBank[245].sName := ' Additional control device information (lockable)';
	aMemoryBank[246].sName := ' Additional control device information (lockable)';
	aMemoryBank[247].sName := ' Additional control device information (lockable)';
	aMemoryBank[248].sName := ' Additional control device information (lockable)';
	aMemoryBank[249].sName := ' Additional control device information (lockable)';
	aMemoryBank[250].sName := ' Additional control device information (lockable)';
	aMemoryBank[251].sName := ' Additional control device information (lockable)';
	aMemoryBank[252].sName := ' Additional control device information (lockable)';
	aMemoryBank[253].sName := ' Additional control device information (lockable)';
	aMemoryBank[254].sName := ' Additional control device information (lockable)';
END_IF
IF (nMemoryBank >= 2) THEN
	aMemoryBank[0].sName := ' Address of last accessible memory location (read only)';
	aMemoryBank[1].sName := ' Indicator byte (manufacturer defined) ';
	aMemoryBank[2].sName := ' Memory bank lock byte';
	aMemoryBank[3].sName := ' Additional control device information (lockable)';
	aMemoryBank[4].sName := ' Additional control device information (lockable)';
	aMemoryBank[5].sName := ' Additional control device information (lockable)';
	aMemoryBank[6].sName := ' Additional control device information (lockable)';
	aMemoryBank[7].sName := ' Additional control device information (lockable)';
	aMemoryBank[8].sName := ' Additional control device information (lockable)';
	aMemoryBank[9].sName := ' Additional control device information (lockable)';
	aMemoryBank[10].sName := ' Additional control device information (lockable)';
	aMemoryBank[11].sName := ' Additional control device information (lockable)';
	aMemoryBank[12].sName := ' Additional control device information (lockable)';
	aMemoryBank[13].sName := ' Additional control device information (lockable)';
	aMemoryBank[14].sName := ' Additional control device information (lockable)';
	aMemoryBank[15].sName := ' Additional control device information (lockable)';
	aMemoryBank[16].sName := ' Additional control device information (lockable)';
END_IF

END_FUNCTION_BLOCK

// ---- Tc3_DALI_PLC_Commissioning_Tool/POUs/DALI_PLC_Commissioning/FB_Part102SetFading.TcPOU
FUNCTION_BLOCK FB_Part102SetFading
VAR_INPUT
	ipDALICommunication			:	I_DALICommunication;
END_VAR
VAR_OUTPUT
	bBusy						:	BOOL;
END_VAR
VAR
	{region "Visu"}
	eAddressType				:	E_DALIAddressType;
	nShortAddress				:	BYTE := 255;
	nGroupAddress				:	BYTE := 255;

	eExtendedFadeTime			:	E_DALIExtendedFadeTime;
	eFadeRate					:	E_DALIFadeRate;
	eFadeTime					:	E_DALIFadeTime;
	bWriteFadeTime				:	BOOL;
	bWriteFadeRate				:	BOOL;
	bWriteExtendedFadeTime		:	BOOL;
	bRead						:	BOOL;
	bHideWaitSymbol				:	BOOL := TRUE;
	{endregion}
	nAddress					:	BYTE;
	nStep						:	INT;
	bNoFadeTime					:	BOOL;

	eExtendedFadeTimeBase		:	E_DALIExtendedFadeTimeBase := E_DALIExtendedFadeTimeBase.Unknown;
	eExtendedFadeTimeMultiplier	:	E_DALIExtendedFadeTimeMultiplier := E_DALIExtendedFadeTimeMultiplier.Unknown;

	fbSetExtendedFadeTime		:	FB_DALI102SetExtendedFadeTime(0);
	fbSetFadeRate				:	FB_DALI102SetFadeRate(0);
	fbSetFadeTime				:	FB_DALI102SetFadeTime(0);

	fbQueryExtendedFadeTime		:	FB_DALI102QueryExtendedFadeTime(0);
	fbQueryFadeTimeFadeRate		:	FB_DALI102QueryFadeTimeFadeRate(0);
END_VAR

{region "Detect Commands"}
IF (bRead AND (nStep =0)) then
	nStep := 10;
	bRead := FALSE;
	bHideWaitSymbol := FALSE;
END_IF
IF (bWriteFadeTime AND (nStep = 0)) THEN
	nStep := 1000;
	bWriteFadeTime := FALSE;
	bHideWaitSymbol := FALSE;
END_IF

IF (bWriteFadeRate AND (nStep = 0)) THEN
	nStep := 1010;
	bWriteFadeRate := FALSE;
	bHideWaitSymbol := FALSE;
END_IF
	 
IF (bWriteExtendedFadeTime AND (nStep = 0) AND (eFadeTime = E_DALIFadeTime.Disabled)) THEN
	nStep := 1020;
	bWriteExtendedFadeTime := FALSE;
	bHideWaitSymbol := FALSE;
END_IF
{endregion}

{region "Manage Dialog Selection"}
IF (nStep = 0) THEN
	bBusy := FALSE;
ELSE
	bBusy := TRUE;
END_IF
{endregion}
nAddress := SEL(eAddressType = E_DALIAddressType.Short, nGroupAddress, nShortAddress);
{region "Execute Commands"}
CASE nStep OF
0:
{region "Init"}
	bWriteFadeTime := FALSE;
	bWriteFadeRate := FALSE;
	bWriteExtendedFadeTime := FALSE;
	bHideWaitSymbol := TRUE;

	fbQueryExtendedFadeTime.ipDALICommunication := ipDALICommunication;
	fbQueryFadeTimeFadeRate.ipDALICommunication := ipDALICommunication;

	fbSetExtendedFadeTime.ipDALICommunication := ipDALICommunication;
	fbSetFadeRate.ipDALICommunication := ipDALICommunication;
	fbSetFadeTime.ipDALICommunication := ipDALICommunication;
{endregion}
10:
{region "Query Fade Time and Fade Rate"}
	fbQueryFadeTimeFadeRate(bStart := TRUE,
							nAddress := nAddress,
							eAddressType := eAddressType,
							eCommandPriority := E_DALICommandPriority.Middle,
							eFadeTime=> eFadeTime,
							eFadeRate=> eFadeRate);
	IF (NOT fbQueryFadeTimeFadeRate.bBusy) THEN
		fbQueryFadeTimeFadeRate(bStart := FALSE);
		IF (eFadeTime = 0) THEN 
			bNoFadeTime := FALSE; // Check whether Fade Time is available
			nStep := 20;
		ELSE 	 
			bNoFadeTime := TRUE;
			nStep := 0;
		END_IF
	END_IF
{endregion}
20:
{region "Query Extended Fade Time"}
	fbQueryExtendedFadeTime(bStart := TRUE,
							nAddress := nAddress,
							eAddressType := eAddressType,
							eCommandPriority := E_DALICommandPriority.Middle,
							eExtendedFadeTimeBase=> eExtendedFadeTimeBase,
							eExtendedFadeTimeMultiplier=> eExtendedFadeTimeMultiplier);
	IF (NOT fbQueryExtendedFadeTime.bBusy) THEN
		fbQueryExtendedFadeTime(bStart := FALSE);
		nStep := 0;
		IF (eExtendedFadeTimeMultiplier = E_DALIExtendedFadeTimeMultiplier.Disabled) THEN
			eExtendedFadeTime := E_DALIExtendedFadeTime.NoFade;
		END_IF
		IF (eExtendedFadeTimeMultiplier = E_DALIExtendedFadeTimeMultiplier.Multiplier100ms) THEN
			CASE eExtendedFadeTimeBase OF
				E_DALIExtendedFadeTimeBase.Base01:	eExtendedFadeTime := E_DALIExtendedFadeTime.onehundred;
				E_DALIExtendedFadeTimeBase.Base02:	eExtendedFadeTime := E_DALIExtendedFadeTime.twohundred;
				E_DALIExtendedFadeTimeBase.Base03:	eExtendedFadeTime := E_DALIExtendedFadeTime.threehundred;
				E_DALIExtendedFadeTimeBase.Base04:	eExtendedFadeTime := E_DALIExtendedFadeTime.fourhundred;
				E_DALIExtendedFadeTimeBase.Base05:	eExtendedFadeTime := E_DALIExtendedFadeTime.fivehundred;
				E_DALIExtendedFadeTimeBase.Base06:	eExtendedFadeTime := E_DALIExtendedFadeTime.sixhundred;
				E_DALIExtendedFadeTimeBase.Base07:	eExtendedFadeTime := E_DALIExtendedFadeTime.sevenhundred;
				E_DALIExtendedFadeTimeBase.Base08:	eExtendedFadeTime := E_DALIExtendedFadeTime.eighthundred;
				E_DALIExtendedFadeTimeBase.Base09:	eExtendedFadeTime := E_DALIExtendedFadeTime.ninehundred;
				E_DALIExtendedFadeTimeBase.Base10:	eExtendedFadeTime := E_DALIExtendedFadeTime.onethousand;
				E_DALIExtendedFadeTimeBase.Base11:	eExtendedFadeTime := E_DALIExtendedFadeTime.onethousandonehundred;
				E_DALIExtendedFadeTimeBase.Base12:	eExtendedFadeTime := E_DALIExtendedFadeTime.onethousandtwohundred;
				E_DALIExtendedFadeTimeBase.Base13:	eExtendedFadeTime := E_DALIExtendedFadeTime.onethousandthreehundred;
				E_DALIExtendedFadeTimeBase.Base14:	eExtendedFadeTime := E_DALIExtendedFadeTime.onethousandfourhundred;
				E_DALIExtendedFadeTimeBase.Base15:	eExtendedFadeTime := E_DALIExtendedFadeTime.onethousandfivehundred;
				E_DALIExtendedFadeTimeBase.Base16:	eExtendedFadeTime := E_DALIExtendedFadeTime.onethousandsixhundred;
			END_CASE
		END_IF
	 	IF (eExtendedFadeTimeMultiplier = E_DALIExtendedFadeTimeMultiplier.Multiplier1s) THEN
			CASE eExtendedFadeTimeBase OF
				E_DALIExtendedFadeTimeBase.Base01:	eExtendedFadeTime := E_DALIExtendedFadeTime.onesecond;
				E_DALIExtendedFadeTimeBase.Base02:	eExtendedFadeTime := E_DALIExtendedFadeTime.twoseconds;
				E_DALIExtendedFadeTimeBase.Base03:	eExtendedFadeTime := E_DALIExtendedFadeTime.threeseconds;
				E_DALIExtendedFadeTimeBase.Base04:	eExtendedFadeTime := E_DALIExtendedFadeTime.fourseconds;
				E_DALIExtendedFadeTimeBase.Base05:	eExtendedFadeTime := E_DALIExtendedFadeTime.fiveseconds;
				E_DALIExtendedFadeTimeBase.Base06:	eExtendedFadeTime := E_DALIExtendedFadeTime.sixseconds;
				E_DALIExtendedFadeTimeBase.Base07:	eExtendedFadeTime := E_DALIExtendedFadeTime.sevenseconds;
				E_DALIExtendedFadeTimeBase.Base08:	eExtendedFadeTime := E_DALIExtendedFadeTime.eightseconds;
				E_DALIExtendedFadeTimeBase.Base09:	eExtendedFadeTime := E_DALIExtendedFadeTime.nineseconds;
				E_DALIExtendedFadeTimeBase.Base10:	eExtendedFadeTime := E_DALIExtendedFadeTime.tenseconds;
				E_DALIExtendedFadeTimeBase.Base11:	eExtendedFadeTime := E_DALIExtendedFadeTime.elevenseconds;
				E_DALIExtendedFadeTimeBase.Base12:	eExtendedFadeTime := E_DALIExtendedFadeTime.twelveseconds;
				E_DALIExtendedFadeTimeBase.Base13:	eExtendedFadeTime := E_DALIExtendedFadeTime.thirteenseconds;
				E_DALIExtendedFadeTimeBase.Base14:	eExtendedFadeTime := E_DALIExtendedFadeTime.fourteenseconds;
				E_DALIExtendedFadeTimeBase.Base15:	eExtendedFadeTime := E_DALIExtendedFadeTime.fifteenseconds;
				E_DALIExtendedFadeTimeBase.Base16:	eExtendedFadeTime := E_DALIExtendedFadeTime.sixteenseconds;
			END_CASE
		END_IF
		IF (eExtendedFadeTimeMultiplier = E_DALIExtendedFadeTimeMultiplier.Multiplier10s) THEN
			CASE eExtendedFadeTimeBase OF
				E_DALIExtendedFadeTimeBase.Base01:	eExtendedFadeTime := E_DALIExtendedFadeTime.ten1seconds;
				E_DALIExtendedFadeTimeBase.Base02:	eExtendedFadeTime := E_DALIExtendedFadeTime.twentyseconds;
				E_DALIExtendedFadeTimeBase.Base03:	eExtendedFadeTime := E_DALIExtendedFadeTime.thirtyseconds;
				E_DALIExtendedFadeTimeBase.Base04:	eExtendedFadeTime := E_DALIExtendedFadeTime.fourtyseconds;
				E_DALIExtendedFadeTimeBase.Base05:	eExtendedFadeTime := E_DALIExtendedFadeTime.fiftyseconds;
				E_DALIExtendedFadeTimeBase.Base06:	eExtendedFadeTime := E_DALIExtendedFadeTime.sixtyseconds;
				E_DALIExtendedFadeTimeBase.Base07:	eExtendedFadeTime := E_DALIExtendedFadeTime.seventyseconds;
				E_DALIExtendedFadeTimeBase.Base08:	eExtendedFadeTime := E_DALIExtendedFadeTime.eightyseconds;
				E_DALIExtendedFadeTimeBase.Base09:	eExtendedFadeTime := E_DALIExtendedFadeTime.ninetyseconds;
				E_DALIExtendedFadeTimeBase.Base10:	eExtendedFadeTime := E_DALIExtendedFadeTime.onehundredseconds;
				E_DALIExtendedFadeTimeBase.Base11:	eExtendedFadeTime := E_DALIExtendedFadeTime.onehundredtenseconds;
				E_DALIExtendedFadeTimeBase.Base12:	eExtendedFadeTime := E_DALIExtendedFadeTime.onehundredtwentyseconds;
				E_DALIExtendedFadeTimeBase.Base13:	eExtendedFadeTime := E_DALIExtendedFadeTime.onehundredthirtyseconds;
				E_DALIExtendedFadeTimeBase.Base14:	eExtendedFadeTime := E_DALIExtendedFadeTime.onehundredfourtyseconds;
				E_DALIExtendedFadeTimeBase.Base15:	eExtendedFadeTime := E_DALIExtendedFadeTime.onehundredfiftyseconds;
				E_DALIExtendedFadeTimeBase.Base16:	eExtendedFadeTime := E_DALIExtendedFadeTime.onehundredsixtyseconds;
			END_CASE
		END_IF
		IF (eExtendedFadeTimeMultiplier = E_DALIExtendedFadeTimeMultiplier.Multiplier1min) THEN
			CASE eExtendedFadeTimeBase OF
				E_DALIExtendedFadeTimeBase.Base01:	eExtendedFadeTime := E_DALIExtendedFadeTime.oneminute;
				E_DALIExtendedFadeTimeBase.Base02:	eExtendedFadeTime := E_DALIExtendedFadeTime.twominutes;
				E_DALIExtendedFadeTimeBase.Base03:	eExtendedFadeTime := E_DALIExtendedFadeTime.threeminutes;
				E_DALIExtendedFadeTimeBase.Base04:	eExtendedFadeTime := E_DALIExtendedFadeTime.fourminutes;
				E_DALIExtendedFadeTimeBase.Base05:	eExtendedFadeTime := E_DALIExtendedFadeTime.fiveminutes;
				E_DALIExtendedFadeTimeBase.Base06:	eExtendedFadeTime := E_DALIExtendedFadeTime.sixminutes;
				E_DALIExtendedFadeTimeBase.Base07:	eExtendedFadeTime := E_DALIExtendedFadeTime.sevenminutes;
				E_DALIExtendedFadeTimeBase.Base08:	eExtendedFadeTime := E_DALIExtendedFadeTime.eightminutes;
				E_DALIExtendedFadeTimeBase.Base09:	eExtendedFadeTime := E_DALIExtendedFadeTime.nineminutes;
				E_DALIExtendedFadeTimeBase.Base10:	eExtendedFadeTime := E_DALIExtendedFadeTime.tenminutes;
				E_DALIExtendedFadeTimeBase.Base11:	eExtendedFadeTime := E_DALIExtendedFadeTime.elevenminutes;
				E_DALIExtendedFadeTimeBase.Base12:	eExtendedFadeTime := E_DALIExtendedFadeTime.twelveminutes;
				E_DALIExtendedFadeTimeBase.Base13:	eExtendedFadeTime := E_DALIExtendedFadeTime.thirteenminutes;
				E_DALIExtendedFadeTimeBase.Base14:	eExtendedFadeTime := E_DALIExtendedFadeTime.fourteenminutes;
				E_DALIExtendedFadeTimeBase.Base15:	eExtendedFadeTime := E_DALIExtendedFadeTime.fifteenminutes;
				E_DALIExtendedFadeTimeBase.Base16:	eExtendedFadeTime := E_DALIExtendedFadeTime.sixteenminutes;
			END_CASE
		END_IF
	ELSE
		eExtendedFadeTime := E_DALIExtendedFadeTime.unknown;
	END_IF
{endregion}
1000:
{region "Set Fade Time"}
	fbSetFadeTime(bStart:= TRUE,
				  nAddress:= nAddress,
				  eAddressType := eAddressType,
				  eCommandPriority := E_DALICommandPriority.Middle,
				  eFadeTime := eFadeTime);
	IF (NOT fbSetFadeTime.bBusy) THEN
		fbSetFadeTime(bStart := FALSE);
		{region " Display whether Fade Time is available²}
		IF (eFadeTime = 0) THEN
			bNoFadeTime := FALSE;
		ELSE
			bNoFadeTime := TRUE;
		END_IF
		{endregion}
		nStep := 0;
	END_IF
{endregion}
1010:
{region "Set Fade Rate"}
	fbSetFadeRate(bStart:= TRUE,
				  nAddress:= nAddress,
				  eAddressType := eAddressType,
				  eCommandPriority := E_DALICommandPriority.Middle,
				  eFadeRate := eFadeRate);
	IF (NOT fbSetFadeRate.bBusy) THEN
		fbSetFadeRate(bStart := FALSE);
		nStep := 0;
	END_IF
{endregion}
1020:
{region "Set Extended Fade Time"}
	CASE eExtendedFadeTime OF
		E_DALIExtendedFadeTime.NoFade:					eExtendedFadeTimeBase := E_DALIExtendedFadeTimeBase.Unknown;
														eExtendedFadeTimeMultiplier := E_DALIExtendedFadeTimeMultiplier.Disabled;
		E_DALIExtendedFadeTime.onehundred:				eExtendedFadeTimeBase := E_DALIExtendedFadeTimeBase.Base01;
														eExtendedFadeTimeMultiplier := E_DALIExtendedFadeTimeMultiplier.Multiplier100ms;
		E_DALIExtendedFadeTime.twohundred:				eExtendedFadeTimeBase := E_DALIExtendedFadeTimeBase.Base02;
														eExtendedFadeTimeMultiplier := E_DALIExtendedFadeTimeMultiplier.Multiplier100ms;
		E_DALIExtendedFadeTime.threehundred:			eExtendedFadeTimeBase := E_DALIExtendedFadeTimeBase.Base03;
														eExtendedFadeTimeMultiplier := E_DALIExtendedFadeTimeMultiplier.Multiplier100ms;
		E_DALIExtendedFadeTime.fourhundred:				eExtendedFadeTimeBase := E_DALIExtendedFadeTimeBase.Base04;
														eExtendedFadeTimeMultiplier := E_DALIExtendedFadeTimeMultiplier.Multiplier100ms;
		E_DALIExtendedFadeTime.fivehundred:				eExtendedFadeTimeBase := E_DALIExtendedFadeTimeBase.Base05;
														eExtendedFadeTimeMultiplier := E_DALIExtendedFadeTimeMultiplier.Multiplier100ms;
		E_DALIExtendedFadeTime.sixhundred:				eExtendedFadeTimeBase := E_DALIExtendedFadeTimeBase.Base06;
														eExtendedFadeTimeMultiplier := E_DALIExtendedFadeTimeMultiplier.Multiplier100ms;
		E_DALIExtendedFadeTime.sevenhundred:			eExtendedFadeTimeBase := E_DALIExtendedFadeTimeBase.Base07;
														eExtendedFadeTimeMultiplier := E_DALIExtendedFadeTimeMultiplier.Multiplier100ms;
		E_DALIExtendedFadeTime.eighthundred:			eExtendedFadeTimeBase := E_DALIExtendedFadeTimeBase.Base08;
														eExtendedFadeTimeMultiplier := E_DALIExtendedFadeTimeMultiplier.Multiplier100ms;
		E_DALIExtendedFadeTime.ninehundred:				eExtendedFadeTimeBase := E_DALIExtendedFadeTimeBase.Base09;
														eExtendedFadeTimeMultiplier := E_DALIExtendedFadeTimeMultiplier.Multiplier100ms;
		E_DALIExtendedFadeTime.onethousand:				eExtendedFadeTimeBase := E_DALIExtendedFadeTimeBase.Base10;
														eExtendedFadeTimeMultiplier := E_DALIExtendedFadeTimeMultiplier.Multiplier100ms;
		E_DALIExtendedFadeTime.onethousandonehundred:	eExtendedFadeTimeBase := E_DALIExtendedFadeTimeBase.Base11;
														eExtendedFadeTimeMultiplier := E_DALIExtendedFadeTimeMultiplier.Multiplier100ms;
		E_DALIExtendedFadeTime.onethousandtwohundred:	eExtendedFadeTimeBase := E_DALIExtendedFadeTimeBase.Base12;
														eExtendedFadeTimeMultiplier := E_DALIExtendedFadeTimeMultiplier.Multiplier100ms;
		E_DALIExtendedFadeTime.onethousandthreehundred:	eExtendedFadeTimeBase := E_DALIExtendedFadeTimeBase.Base13;
														eExtendedFadeTimeMultiplier := E_DALIExtendedFadeTimeMultiplier.Multiplier100ms;
		E_DALIExtendedFadeTime.onethousandfourhundred:	eExtendedFadeTimeBase := E_DALIExtendedFadeTimeBase.Base14;
														eExtendedFadeTimeMultiplier := E_DALIExtendedFadeTimeMultiplier.Multiplier100ms;
		E_DALIExtendedFadeTime.onethousandfivehundred:	eExtendedFadeTimeBase := E_DALIExtendedFadeTimeBase.Base15;
														eExtendedFadeTimeMultiplier := E_DALIExtendedFadeTimeMultiplier.Multiplier100ms;
		E_DALIExtendedFadeTime.onethousandsixhundred:	eExtendedFadeTimeBase := E_DALIExtendedFadeTimeBase.Base16;
														eExtendedFadeTimeMultiplier := E_DALIExtendedFadeTimeMultiplier.Multiplier100ms;
		E_DALIExtendedFadeTime.onesecond:				eExtendedFadeTimeBase := E_DALIExtendedFadeTimeBase.Base01;
														eExtendedFadeTimeMultiplier := E_DALIExtendedFadeTimeMultiplier.Multiplier1s;
		E_DALIExtendedFadeTime.twoseconds:				eExtendedFadeTimeBase := E_DALIExtendedFadeTimeBase.Base02;
														eExtendedFadeTimeMultiplier := E_DALIExtendedFadeTimeMultiplier.Multiplier1s;
		E_DALIExtendedFadeTime.threeseconds:			eExtendedFadeTimeBase := E_DALIExtendedFadeTimeBase.Base03;
														eExtendedFadeTimeMultiplier := E_DALIExtendedFadeTimeMultiplier.Multiplier1s;
		E_DALIExtendedFadeTime.fourseconds:				eExtendedFadeTimeBase := E_DALIExtendedFadeTimeBase.Base04;
														eExtendedFadeTimeMultiplier := E_DALIExtendedFadeTimeMultiplier.Multiplier1s;
		E_DALIExtendedFadeTime.fiveseconds:				eExtendedFadeTimeBase := E_DALIExtendedFadeTimeBase.Base05;
														eExtendedFadeTimeMultiplier := E_DALIExtendedFadeTimeMultiplier.Multiplier1s;
		E_DALIExtendedFadeTime.sixseconds:				eExtendedFadeTimeBase := E_DALIExtendedFadeTimeBase.Base06;
														eExtendedFadeTimeMultiplier := E_DALIExtendedFadeTimeMultiplier.Multiplier1s;
		E_DALIExtendedFadeTime.sevenseconds:			eExtendedFadeTimeBase := E_DALIExtendedFadeTimeBase.Base07;
														eExtendedFadeTimeMultiplier := E_DALIExtendedFadeTimeMultiplier.Multiplier1s;
		E_DALIExtendedFadeTime.eightseconds:			eExtendedFadeTimeBase := E_DALIExtendedFadeTimeBase.Base08;
														eExtendedFadeTimeMultiplier := E_DALIExtendedFadeTimeMultiplier.Multiplier1s;
		E_DALIExtendedFadeTime.nineseconds:				eExtendedFadeTimeBase := E_DALIExtendedFadeTimeBase.Base09;
														eExtendedFadeTimeMultiplier := E_DALIExtendedFadeTimeMultiplier.Multiplier1s;
		E_DALIExtendedFadeTime.tenseconds:				eExtendedFadeTimeBase := E_DALIExtendedFadeTimeBase.Base10;
														eExtendedFadeTimeMultiplier := E_DALIExtendedFadeTimeMultiplier.Multiplier1s;
		E_DALIExtendedFadeTime.elevenseconds:			eExtendedFadeTimeBase := E_DALIExtendedFadeTimeBase.Base11;
														eExtendedFadeTimeMultiplier := E_DALIExtendedFadeTimeMultiplier.Multiplier1s;
		E_DALIExtendedFadeTime.twelveseconds:			eExtendedFadeTimeBase := E_DALIExtendedFadeTimeBase.Base12;
														eExtendedFadeTimeMultiplier := E_DALIExtendedFadeTimeMultiplier.Multiplier1s;
		E_DALIExtendedFadeTime.thirteenseconds:			eExtendedFadeTimeBase := E_DALIExtendedFadeTimeBase.Base13;
														eExtendedFadeTimeMultiplier := E_DALIExtendedFadeTimeMultiplier.Multiplier1s;
		E_DALIExtendedFadeTime.fourteenseconds:			eExtendedFadeTimeBase := E_DALIExtendedFadeTimeBase.Base14;
														eExtendedFadeTimeMultiplier := E_DALIExtendedFadeTimeMultiplier.Multiplier1s;
		E_DALIExtendedFadeTime.fifteenseconds:			eExtendedFadeTimeBase := E_DALIExtendedFadeTimeBase.Base15;
														eExtendedFadeTimeMultiplier := E_DALIExtendedFadeTimeMultiplier.Multiplier1s;
		E_DALIExtendedFadeTime.sixteenseconds:			eExtendedFadeTimeBase := E_DALIExtendedFadeTimeBase.Base16;
														eExtendedFadeTimeMultiplier := E_DALIExtendedFadeTimeMultiplier.Multiplier1s;
		E_DALIExtendedFadeTime.ten1seconds:				eExtendedFadeTimeBase := E_DALIExtendedFadeTimeBase.Base01;
														eExtendedFadeTimeMultiplier := E_DALIExtendedFadeTimeMultiplier.Multiplier10s;
		E_DALIExtendedFadeTime.twentyseconds:			eExtendedFadeTimeBase := E_DALIExtendedFadeTimeBase.Base02;
														eExtendedFadeTimeMultiplier := E_DALIExtendedFadeTimeMultiplier.Multiplier10s;
		E_DALIExtendedFadeTime.thirtyseconds:			eExtendedFadeTimeBase := E_DALIExtendedFadeTimeBase.Base03;
														eExtendedFadeTimeMultiplier := E_DALIExtendedFadeTimeMultiplier.Multiplier10s;
		E_DALIExtendedFadeTime.fourtyseconds:			eExtendedFadeTimeBase := E_DALIExtendedFadeTimeBase.Base04;
														eExtendedFadeTimeMultiplier := E_DALIExtendedFadeTimeMultiplier.Multiplier10s;
		E_DALIExtendedFadeTime.fiftyseconds:			eExtendedFadeTimeBase := E_DALIExtendedFadeTimeBase.Base05;
														eExtendedFadeTimeMultiplier := E_DALIExtendedFadeTimeMultiplier.Multiplier10s;
		E_DALIExtendedFadeTime.sixtyseconds:			eExtendedFadeTimeBase := E_DALIExtendedFadeTimeBase.Base06;
														eExtendedFadeTimeMultiplier := E_DALIExtendedFadeTimeMultiplier.Multiplier10s;
		E_DALIExtendedFadeTime.seventyseconds:			eExtendedFadeTimeBase := E_DALIExtendedFadeTimeBase.Base07;
														eExtendedFadeTimeMultiplier := E_DALIExtendedFadeTimeMultiplier.Multiplier10s;
		E_DALIExtendedFadeTime.eightyseconds:			eExtendedFadeTimeBase := E_DALIExtendedFadeTimeBase.Base08;
														eExtendedFadeTimeMultiplier := E_DALIExtendedFadeTimeMultiplier.Multiplier10s;
		E_DALIExtendedFadeTime.ninetyseconds:			eExtendedFadeTimeBase := E_DALIExtendedFadeTimeBase.Base09;
														eExtendedFadeTimeMultiplier := E_DALIExtendedFadeTimeMultiplier.Multiplier10s;
		E_DALIExtendedFadeTime.onehundredseconds:		eExtendedFadeTimeBase := E_DALIExtendedFadeTimeBase.Base10;
														eExtendedFadeTimeMultiplier := E_DALIExtendedFadeTimeMultiplier.Multiplier10s;
		E_DALIExtendedFadeTime.onehundredtenseconds:	eExtendedFadeTimeBase := E_DALIExtendedFadeTimeBase.Base11;
														eExtendedFadeTimeMultiplier := E_DALIExtendedFadeTimeMultiplier.Multiplier10s;
		E_DALIExtendedFadeTime.onehundredtwentyseconds:	eExtendedFadeTimeBase := E_DALIExtendedFadeTimeBase.Base12;
														eExtendedFadeTimeMultiplier := E_DALIExtendedFadeTimeMultiplier.Multiplier10s;
		E_DALIExtendedFadeTime.onehundredthirtyseconds:	eExtendedFadeTimeBase := E_DALIExtendedFadeTimeBase.Base13;
														eExtendedFadeTimeMultiplier := E_DALIExtendedFadeTimeMultiplier.Multiplier10s;
		E_DALIExtendedFadeTime.onehundredfourtyseconds:	eExtendedFadeTimeBase := E_DALIExtendedFadeTimeBase.Base14;
														eExtendedFadeTimeMultiplier := E_DALIExtendedFadeTimeMultiplier.Multiplier10s;
		E_DALIExtendedFadeTime.onehundredfiftyseconds:	eExtendedFadeTimeBase := E_DALIExtendedFadeTimeBase.Base15;
														eExtendedFadeTimeMultiplier := E_DALIExtendedFadeTimeMultiplier.Multiplier10s;
		E_DALIExtendedFadeTime.onehundredsixtyseconds:	eExtendedFadeTimeBase := E_DALIExtendedFadeTimeBase.Base16;
														eExtendedFadeTimeMultiplier := E_DALIExtendedFadeTimeMultiplier.Multiplier10s;
		E_DALIExtendedFadeTime.oneminute:				eExtendedFadeTimeBase := E_DALIExtendedFadeTimeBase.Base01;
														eExtendedFadeTimeMultiplier := E_DALIExtendedFadeTimeMultiplier.Multiplier1min;
		E_DALIExtendedFadeTime.twominutes:				eExtendedFadeTimeBase := E_DALIExtendedFadeTimeBase.Base02;
														eExtendedFadeTimeMultiplier := E_DALIExtendedFadeTimeMultiplier.Multiplier1min;
		E_DALIExtendedFadeTime.threeminutes:			eExtendedFadeTimeBase := E_DALIExtendedFadeTimeBase.Base03;
														eExtendedFadeTimeMultiplier := E_DALIExtendedFadeTimeMultiplier.Multiplier1min;
		E_DALIExtendedFadeTime.fourminutes:				eExtendedFadeTimeBase := E_DALIExtendedFadeTimeBase.Base04;
														eExtendedFadeTimeMultiplier := E_DALIExtendedFadeTimeMultiplier.Multiplier1min;
		E_DALIExtendedFadeTime.fiveminutes:				eExtendedFadeTimeBase := E_DALIExtendedFadeTimeBase.Base05;
														eExtendedFadeTimeMultiplier := E_DALIExtendedFadeTimeMultiplier.Multiplier1min;
		E_DALIExtendedFadeTime.sixminutes:				eExtendedFadeTimeBase := E_DALIExtendedFadeTimeBase.Base06;
														eExtendedFadeTimeMultiplier := E_DALIExtendedFadeTimeMultiplier.Multiplier1min;
		E_DALIExtendedFadeTime.sevenminutes:			eExtendedFadeTimeBase := E_DALIExtendedFadeTimeBase.Base07;
														eExtendedFadeTimeMultiplier := E_DALIExtendedFadeTimeMultiplier.Multiplier1min;
		E_DALIExtendedFadeTime.eightminutes:			eExtendedFadeTimeBase := E_DALIExtendedFadeTimeBase.Base08;
														eExtendedFadeTimeMultiplier := E_DALIExtendedFadeTimeMultiplier.Multiplier1min;
		E_DALIExtendedFadeTime.nineminutes:				eExtendedFadeTimeBase := E_DALIExtendedFadeTimeBase.Base09;
														eExtendedFadeTimeMultiplier := E_DALIExtendedFadeTimeMultiplier.Multiplier1min;
		E_DALIExtendedFadeTime.tenminutes:				eExtendedFadeTimeBase := E_DALIExtendedFadeTimeBase.Base10;
														eExtendedFadeTimeMultiplier := E_DALIExtendedFadeTimeMultiplier.Multiplier1min;
		E_DALIExtendedFadeTime.elevenminutes:			eExtendedFadeTimeBase := E_DALIExtendedFadeTimeBase.Base11;
														eExtendedFadeTimeMultiplier := E_DALIExtendedFadeTimeMultiplier.Multiplier1min;
		E_DALIExtendedFadeTime.twelveminutes:			eExtendedFadeTimeBase := E_DALIExtendedFadeTimeBase.Base12;
														eExtendedFadeTimeMultiplier := E_DALIExtendedFadeTimeMultiplier.Multiplier1min;
		E_DALIExtendedFadeTime.thirteenminutes:			eExtendedFadeTimeBase := E_DALIExtendedFadeTimeBase.Base13;
														eExtendedFadeTimeMultiplier := E_DALIExtendedFadeTimeMultiplier.Multiplier1min;
		E_DALIExtendedFadeTime.fourteenminutes:			eExtendedFadeTimeBase := E_DALIExtendedFadeTimeBase.Base14;
														eExtendedFadeTimeMultiplier := E_DALIExtendedFadeTimeMultiplier.Multiplier1min;
		E_DALIExtendedFadeTime.fifteenminutes:			eExtendedFadeTimeBase := E_DALIExtendedFadeTimeBase.Base15;
														eExtendedFadeTimeMultiplier := E_DALIExtendedFadeTimeMultiplier.Multiplier1min;
		E_DALIExtendedFadeTime.sixteenminutes:			eExtendedFadeTimeBase := E_DALIExtendedFadeTimeBase.Base16;
														eExtendedFadeTimeMultiplier := E_DALIExtendedFadeTimeMultiplier.Multiplier1min;
		E_DALIExtendedFadeTime.unknown:					eExtendedFadeTimeBase := E_DALIExtendedFadeTimeBase.Unknown;
														eExtendedFadeTimeMultiplier := E_DALIExtendedFadeTimeMultiplier.Unknown;
	END_CASE
	fbSetExtendedFadeTime(bStart:= TRUE,
						  nAddress:= nAddress,
						  eAddressType := eAddressType,
						  eCommandPriority := E_DALICommandPriority.Middle,
						  eExtendedFadeTimeBase := eExtendedFadeTimeBase,
						  eExtendedFadeTimeMultiplier := eExtendedFadeTimeMultiplier);
	IF (NOT fbSetExtendedFadeTime.bBusy) THEN
		fbSetExtendedFadeTime(bStart := FALSE);
		nStep := 0;
	END_IF
{endregion}
END_CASE

END_FUNCTION_BLOCK

// ---- Bridge/FB_DALIBridge.TcPOU
FUNCTION_BLOCK FB_DALIBridge
VAR_INPUT
	// On rising edge, initialises the function block.
	initialise				: BOOL := TRUE;
	emergency				: BOOL := FALSE;
END_VAR
VAR_OUTPUT
	// RPC client will watch for changes to this variable
	// it contains the result of the last completed request
	rpcResponse            	: ST_DALIBridgeResponse;
	// RPC client will watch for changes to this to be notified about
	// events that have occurred
	notification            : ST_DALIBridgeNotification;
END_VAR
VAR
	rtrigInitialise				: R_TRIG;
	
	// internal request handling state
	requestFirstCycle       	: BOOL; 				// TRUE if this is the first cycle of a new request
													// used to create a rising edge on the start of a request
	activeRequest				: ST_DALIBridgeRequest;	// request being processed currently
	activeRequestSequence   	: ULINT;				// sequence number of the current request
	requestCounter          	: ULINT := 1;			// incremented to generate sequence numbers for requests

	// notification handling
	notificationAcked       	: BOOL := TRUE;			// true if it is OK to send a new notification
	notificationCounter     	: ULINT := 1;
	
	// DALI command function blocks
	communication				: I_DALICommunication := 0;
	fbEmergencyPowerOn			: FB_DALI102RecallMaxLevel(0);
	fbDirectArcPowerControl 	: FB_DALI102DirectArcPowerControl(0);
	fbQueryActualLevel      	: FB_DALI102QueryActualLevel(0);
	fbQueryStatus           	: FB_DALI102QueryStatus(0);
	fbSetEventScheme        	: FB_DALI103SetEventScheme(0);
	fbQueryEventScheme      	: FB_DALI103QueryEventScheme(0);
	fbSetEventFilter        	: FB_DALI103SetEventFilter(0);
	fbQueryEventFilter      	: FB_DALI103QueryEventFilter(0);
	fbIdentifyDevice102     	: FB_DALI102IdentifyDevice(0);
	fbIdentifyDevice103     	: FB_DALI103IdentifyDevice(0);
	fbEnableInstance        	: FB_DALI103EnableInstance(0);
	fbGoToScene					: FB_DALI102GoToScene(0);
	fbSetFadeTime 				: FB_DALI102SetFadeTime(0);
	fbQueryInputValue			: FB_DALI103QueryInputValue(0);
	fbQueryBatteryCharge        : FB_DALI202QueryBatteryCharge(0);
	fbQueryDurationTestResult   : FB_DALI202QueryDurationTestResult(0);
	fbQueryEmergencyMode        : FB_DALI202QueryEmergencyMode(0);
	fbQueryEmergencyStatus      : FB_DALI202QueryEmergencyStatus(0);
	fbQueryFailureStatus        : FB_DALI202QueryFailureStatus(0);
	fbQueryRatedDuration        : FB_DALI202QueryRatedDuration(0);
	fbQueryTestTiming           : FB_DALI202QueryTestTiming(0);
	fbResetDurationTestDoneFlag : FB_DALI202ResetDurationTestDoneFlag(0);
	fbResetFunctionTestDoneFlag : FB_DALI202ResetFunctionTestDoneFlag(0);
	fbStartDurationTest         : FB_DALI202StartDurationTest(0);
	fbStartFunctionTest 		: FB_DALI202StartFunctionTest(0);
	fbStopTest                  : FB_DALI202StopTest(0);
	fbSetDurationTestInterval   : FB_DALI202SetDurationTestInterval(0);
	fbSetFunctionTestInterval   : FB_DALI202SetFunctionTestInterval(0);
	fbStartIdentification202    : FB_DALI202StartIdentification(0);
	fbQueryGroups               : FB_DALI102QueryGroups(0);
	fbAddToGroup				: FB_DALI102AddToGroup(0);
	fbRemoveFromGroup			: FB_DALI102RemoveFromGroup(0);
	
	// input monitor function blocks
	numInputEventListeners  	: INT := 0;
	inputEventListenerParams 	: ARRAY [0..GVL_DALIBridge.maxInputEventListeners-1] OF ST_DALIBridgeInputEventParams;
	fbsGetInputNotification 	: ARRAY [0..GVL_DALIBridge.maxInputEventListeners-1] OF FB_DALIGetInputNotification(0);
	
	// temporary / work variables
	reinterpretEnum				: U_ReinterpretDALIEnum;

END_VAR

// initialise function block when requested
rtrigInitialise( clk := initialise );
IF (rtrigInitialise.Q OR isFirstCycle()) THEN
	ADSLOGSTR(
		msgFmtStr := 'initialise FB_DALIBridge',
		strArg := '',
		msgCtrlMask := ADSLOG_MSGTYPE_LOG
	);
	initCommunication();
	activeRequest.command := E_DALIBridgeCommand.idle;
END_IF

fbEmergencyPowerOn(
	bStart := emergency,
	nAddress := 0,
	eAddressType := E_DALIAddressType.Broadcast,
	eCommandPriority := E_DALICommandPriority.High
);


// work on the active request
CASE activeRequest.command OF
E_DALIBridgeCommand.directArcPowerControl:
	fbDirectArcPowerControl( 
		bStart 				:= requestFirstCycle,
		nAddress 			:= activeRequest.address,
		eAddressType 		:= activeRequest.addressType,
		eCommandPriority 	:= E_DALICommandPriority.Middle,
		nArcPowerLevel		:= activeRequest.data );
	IF emergency THEN
		cancelCommand();
	ELSE
		processResult(
			busy 			:= fbDirectArcPowerControl.bBusy,
			data 			:= 0,
			bError 			:= fbDirectArcPowerControl.bError,
			ipResultMessage := fbDirectArcPowerControl.ipResultMessage
		);
	END_IF;
	
E_DALIBridgeCommand.queryActualLevel:
	fbQueryActualLevel( 
		bStart 				:= requestFirstCycle,
		nAddress 			:= activeRequest.address,
		eAddressType 		:= activeRequest.addressType,
		eCommandPriority 	:= E_DALICommandPriority.Middle );
	processResult(
		busy 			:= fbQueryActualLevel.bBusy,
		data 			:= fbQueryActualLevel.nActualLevel,
		bError 			:= fbQueryActualLevel.bError,
		ipResultMessage := fbQueryActualLevel.ipResultMessage
	);			

E_DALIBridgeCommand.queryStatus:
	fbQueryStatus( 
		bStart 				:= requestFirstCycle,
		nAddress 			:= activeRequest.address,
		eAddressType 		:= activeRequest.addressType,
		eCommandPriority 	:= E_DALICommandPriority.Middle 
	);
	processResult( 
		busy 				:= fbQueryStatus.bBusy,
		bError 				:= fbQueryStatus.bError,
		data 				:= fbQueryStatus.nStatus,
		ipResultMessage 	:= fbQueryStatus.ipResultMessage 
	);	
				   
E_DALIBridgeCommand.setEventScheme:
	// cast the data byte we got to the enum type required
	reinterpretEnum.raw := activeRequest.data;
	fbSetEventScheme(
		bStart 					:= requestFirstCycle,
		nAddress 				:= activeRequest.address,
		eAddressType 			:= activeRequest.addressType,
		nInstanceAddress 		:= activeRequest.instanceAddress,
		eInstanceAddressType 	:= activeRequest.instanceAddressType,
		eEventScheme 			:= reinterpretEnum.eventScheme,
		eCommandPriority 		:= E_DALICommandPriority.Middle,
	);
	processResult(
		busy 			:= fbSetEventScheme.bBusy,
		bError 			:= fbSetEventScheme.bError,
		data   			:= 0,
		ipResultMessage := fbSetEventScheme.ipResultMessage,
	);
	
E_DALIBridgeCommand.queryEventScheme:
	fbQueryEventScheme(
		bStart					:= requestFirstCycle,
		nAddress				:= activeRequest.address,
		eAddressType 			:= activeRequest.addressType,
		nInstanceAddress		:= activeRequest.instanceAddress,
		eInstanceAddressType	:= activeRequest.instanceAddressType,
		eCommandPriority		:= E_DALICommandPriority.Middle
	);
	processResult(
		busy			:= fbQueryEventScheme.bBusy,
		bError			:= fbQueryEventScheme.bError,
		data 			:= fbQueryEventScheme.eEventScheme,
		ipResultMessage := fbQueryEventScheme.ipResultMessage
	);
	
E_DALIBridgeCommand.setEventFilter:
	fbSetEventFilter(
		bStart					:= requestFirstCycle,
		nAddress				:= activeRequest.address,
		eAddressType			:= activeRequest.addressType,
		nInstanceAddress		:= activeRequest.instanceAddress,
		eInstanceAddressType 	:= activeRequest.instanceAddressType,
		nEventFilter 			:= activeRequest.data
	);
	processResult(
		busy			:= fbSetEventFilter.bBusy,
		bError			:= fbSetEventFilter.bError,
		data			:= 0,
		ipResultMessage := fbSetEventFilter.ipResultMessage	
	);

E_DALIBridgeCommand.queryEventFilter:
	fbQueryEventFilter(
		bStart					:= requestFirstCycle,
		nAddress				:= activeRequest.address,
		eAddressType			:= activeRequest.addressType,
		nInstanceAddress		:= activeRequest.instanceAddress,
		eInstanceAddressType	:= activeRequest.instanceAddressType,
		eCommandPriority 		:= E_DALICommandPriority.Middle
	);
	processResult(
		busy			:= fbQueryEventFilter.bBusy,
		bError			:= fbQueryEventFilter.bError,
		data 			:= DWORD_TO_BYTE(fbQueryEventFilter.nEventFilter),
		ipResultMessage := fbQueryEventFilter.ipResultMessage
	);
	
E_DALIBridgeCommand.identifyDevice102:
	fbIdentifyDevice102(
		bStart					:= requestFirstCycle,
		nAddress				:= activeRequest.address,
		eAddressType			:= activeRequest.addressType,
		eCommandPriority		:= E_DALICommandPriority.Middle
	);
	processResult(
		busy			:= fbIdentifyDevice102.bBusy,
		bError			:= fbIdentifyDevice102.bError,
		data 			:= 0,
		ipResultMessage := fbIdentifyDevice102.ipResultMessage
	);
	
E_DALIBridgeCommand.identifyDevice103:
	fbIdentifyDevice103(
		bStart					:= requestFirstCycle,
		nAddress				:= activeRequest.address,
		eAddressType			:= activeRequest.addressType,
		eCommandPriority		:= E_DALICommandPriority.Middle
	);
	processResult(
		busy			:= fbIdentifyDevice103.bBusy,
		bError			:= fbIdentifyDevice103.bError,
		data 			:= 0,
		ipResultMessage := fbIdentifyDevice103.ipResultMessage
	);
	
E_DALIBridgeCommand.enableInstance:
	fbEnableInstance(
		bStart					:= requestFirstCycle,
		nAddress 				:= activeRequest.address,
		eAddressType			:= activeRequest.addressType,
		nInstanceAddress		:= activeRequest.instanceAddress,
		eInstanceAddressType	:= activeRequest.instanceAddressType,
		eCommandPriority 		:= E_DALICommandPriority.Middle
	);
	processResult(
		busy			:= fbEnableInstance.bBusy,
		bError			:= fbEnableInstance.bError,
		data			:= 0,
		ipResultMessage := fbEnableInstance.ipResultMessage
	);
	
E_DALIBridgeCommand.goToScene:
	fbGoToScene(
		bStart 					:= requestFirstCycle,
		nAddress 				:= activeRequest.address,
		eAddressType			:= activeRequest.addressType,
		nScene 					:= activeRequest.data,
		eCommandPriority		:= E_DALICommandPriority.Middle
	);
	IF emergency THEN
		cancelCommand();
	ELSE
		processResult(
			busy			:= fbGoToScene.bBusy,
			bError			:= fbGoToScene.bError,
			data			:= 0,
			ipResultMessage := fbGoToScene.ipResultMessage
		);
	END_IF
	
E_DALIBridgeCommand.setFadeTime:
	reinterpretEnum.raw := activeRequest.data;
	fbSetFadeTime(
		bStart 					:= requestFirstCycle,
		nAddress 				:= activeRequest.address,
		eAddressType			:= activeRequest.addressType,
		eFadeTime 				:= reinterpretEnum.fadeTime
	);
	processResult(
		busy			:= fbSetFadeTime.bBusy,
		bError 			:= fbSetFadeTime.bError,
		data 			:= 0,
		ipResultMessage := fbSetFadeTime.ipResultMessage
	);
	
E_DALIBridgeCommand.queryInputValue:
	fbQueryInputValue(
		bStart					:= requestFirstCycle,
		nAddress				:= activeRequest.address,
		eAddressType			:= activeRequest.addressType,
		nInstanceAddress		:= activeRequest.instanceAddress,
		eInstanceAddressType	:= activeRequest.instanceAddressType,
		nResolution				:= 8,
		eCommandPriority		:= E_DALICommandPriority.Middle
	);
	processResult(
		busy					:= fbQueryInputValue.bBusy,
		bError					:= fbQueryInputValue.bError,
		data					:= fbQueryInputValue.nInputValue,
		ipResultMessage			:= fbQueryInputValue.ipResultMessage
	);
	
E_DALIBridgeCommand.queryBatteryCharge:
	fbQueryBatteryCharge(
		bStart					:= requestFirstCycle,
		nAddress				:= activeRequest.address,
		eAddressType			:= activeRequest.addressType
	);
	processResult(
		busy					:= fbQueryBatteryCharge.bBusy,
		bError					:= fbQueryBatteryCharge.bError,
		data					:= fbQueryBatteryCharge.nBatteryCharge,
		ipResultMessage			:= fbQueryBatteryCharge.ipResultMessage
	);	
	
E_DALIBridgeCommand.queryDurationTestResult:
	fbQueryDurationTestResult(
		bStart					:= requestFirstCycle,
		nAddress				:= activeRequest.address,
		eAddressType			:= activeRequest.addressType
	);
	processResult(
		busy					:= fbQueryDurationTestResult.bBusy,
		bError					:= fbQueryDurationTestResult.bError,
		data					:= fbQueryDurationTestResult.nDurationTestResult,
		ipResultMessage			:= fbQueryDurationTestResult.ipResultMessage
	);	
	
E_DALIBridgeCommand.queryEmergencyMode:
	fbQueryEmergencyMode(
		bStart					:= requestFirstCycle,
		nAddress				:= activeRequest.address,
		eAddressType			:= activeRequest.addressType
	);
	processResult(
		busy					:= fbQueryEmergencyMode.bBusy,
		bError					:= fbQueryEmergencyMode.bError,
		data					:= fbQueryEmergencyMode.nEmergencyMode,
		ipResultMessage			:= fbQueryEmergencyMode.ipResultMessage
	);
	
E_DALIBridgeCommand.queryEmergencyStatus:
	fbQueryEmergencyStatus(
		bStart					:= requestFirstCycle,
		nAddress				:= activeRequest.address,
		eAddressType			:= activeRequest.addressType
	);
	processResult(
		busy					:= fbQueryEmergencyStatus.bBusy,
		bError					:= fbQueryEmergencyStatus.bError,
		data					:= fbQueryEmergencyStatus.nEmergencyStatus,
		ipResultMessage			:= fbQueryEmergencyStatus.ipResultMessage
	);
	
E_DALIBridgeCommand.queryFailureStatus:
	fbQueryFailureStatus(
		bStart					:= requestFirstCycle,
		nAddress				:= activeRequest.address,
		eAddressType			:= activeRequest.addressType
	);
	processResult(
		busy					:= fbQueryFailureStatus.bBusy,
		bError					:= fbQueryFailureStatus.bError,
		data					:= fbQueryFailureStatus.nFailureStatus,
		ipResultMessage			:= fbQueryFailureStatus.ipResultMessage
	);
	
E_DALIBridgeCommand.queryRatedDuration:
	fbQueryRatedDuration(
		bStart					:= requestFirstCycle,
		nAddress				:= activeRequest.address,
		eAddressType			:= activeRequest.addressType
	);
	processResult(
		busy					:= fbQueryRatedDuration.bBusy,
		bError					:= fbQueryRatedDuration.bError,
		data					:= fbQueryRatedDuration.nRatedDuration,
		ipResultMessage			:= fbQueryRatedDuration.ipResultMessage
	);
	
E_DALIBridgeCommand.queryTestTiming:
	reinterpretEnum.raw := activeRequest.data;
	fbQueryTestTiming(
		bStart					:= requestFirstCycle,
		nAddress				:= activeRequest.address,
		eAddressType			:= activeRequest.addressType,
		eTestTiming				:= reinterpretEnum.testTiming
	);
	processResult(
		busy					:= fbQueryTestTiming.bBusy,
		bError					:= fbQueryTestTiming.bError,
		data					:= fbQueryTestTiming.nValue,
		ipResultMessage			:= fbQueryTestTiming.ipResultMessage
	);
	
